KUKA KRL program: EPS_2_25694_CR02_A_20260114065854.src

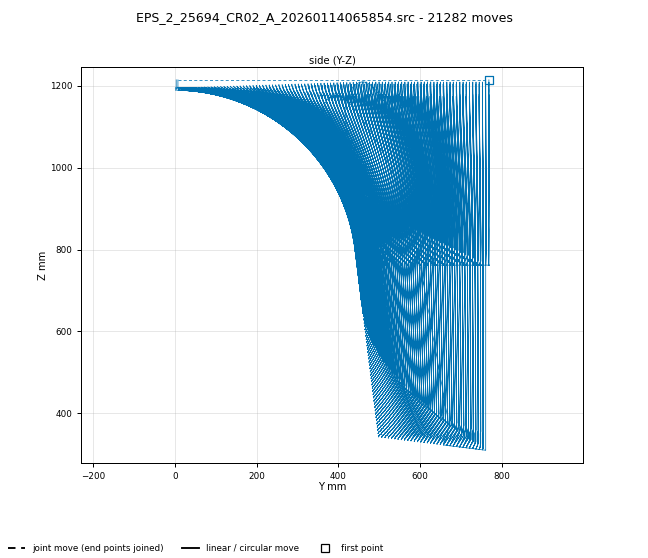
[picture p0: tool path of EPS_2_25694_CR02_A_20260114065854.src, 21282 of 21284 moves have a stored position in this frame; points joined in program order, loops and branches not executed]
&ACCESS RVP
&REL 4
&COMMENT QRS 19112012
&PARAM EDITMASK = *
DEF PART()
EXT BAS (BAS_COMMAND :IN,REAL :IN )
INT I
BAS (#INITMOV,0 )

;KUKA QRS Post kuka4.cps  Date:22-06-2017 !

File_ID=2972

QRS_PRE_INIT()

;Init var - Until changes are made in qrs_pre_init
Outlet_Square_prg=0
Inlet_1_Square_prg=0
Inlet_2_Square_prg=0
Inlet_3_Square_prg=0
Inlet_4_Square_prg=0
Inlet_5_Square_prg=0

Outlet_1={X 0.000, Y 457.000, Z 786.000, B 0.000, E1 0.000 }
Inlet_1={X 0.000, Y 457.000, Z 756.000, B 0.000, E1 180.000 }
Outlet_1_type=838
Inlet_1_type=838
;QRS#1=Sidecore dimensions
;QRS#2=825-33" Concrete
;QRS#3=825-33" Concrete
;QRS#4=
;QRS#5=
;QRS#6=
;QRS#7=
;QRS#8=
;QRS#9=S306-46
;QRS#10=S306-46
;QRS#11=
;QRS#12=
;QRS#13=
;QRS#14=
;QRS#15=
;QRS#16=1524x152x1676 5,5'
;QRS#17=EPS Height
;QRS#18=1205
;QRS#19=*
;QRS#20= UPDATED VERSION 22-06-2017
;QRS#21=*
Outlet_Square=0650
Inlet_1_Square=0650
Inlet_2_Square=0
Inlet_3_Square=0
Inlet_4_Square=0
Inlet_5_Square=0
Mill_Square=1
Outlet_Square_Prg=267
Inlet_1_Square_prg=267

QRS_INIT()

$ADVANCE=5

; T1
PTP {E1 173.011,E2 173.011}
PTP {X 0,Y 767.721,A -85,B 0,C 180,E1 173.011,E2 173.011,E3 0,E4 0,E5 0,E6 0}
QRS_SPEED_INIT()
LIN {X 0,Y 767.721,Z 1215,A -85,B 0,C 180,E1 173.011,E2 173.011,E3 0,E4 0,E5 0,E6 0} C_VEL
LIN {X 0,Y 767.721,Z 764.06,A -85,B 0,C 180,E1 173.011,E2 173.011} C_VEL
LIN {X 0,Y 767.758,Z 762.06,A -85,B 0,C 180,E1 173.16,E2 173.16} C_VEL
LIN {X 0,Y 767.849,Z 762.06,A -85,B 0,C 180,E1 173.458,E2 173.458} C_VEL
LIN {X 0,Y 767.873,Z 762.06,A -85,B 0,C 180,E1 177.201,E2 177.201} C_VEL
LIN {X 0,Y 767.866,Z 762.06,A -85,B 0,C 180,E1 180.933,E2 180.933} C_VEL
LIN {X 0,Y 767.801,Z 762.06,A -85,B 0,C 180,E1 184.668,E2 184.668} C_VEL
LIN {X 0,Y 767.796,Z 762.06,A -85,B 0,C 180,E1 188.424,E2 188.424} C_VEL
LIN {X 0,Y 767.786,Z 762.06,A -85,B 0,C 180,E1 192.216,E2 192.216} C_VEL
LIN {X 0,Y 767.853,Z 762.06,A -85,B 0,C 180,E1 196.217,E2 196.217} C_VEL
LIN {X 0,Y 767.811,Z 762.06,A -85,B 0,C 180,E1 199.987,E2 199.987} C_VEL
LIN {X 0,Y 767.795,Z 762.06,A -85,B 0,C 180,E1 204.011,E2 204.011} C_VEL
LIN {X 0,Y 767.772,Z 762.06,A -85,B 0,C 180,E1 208.166,E2 208.166} C_VEL
LIN {X 0,Y 767.321,Z 762.06,A -85,B 0,C 180,E1 210.327,E2 210.327} C_VEL
LIN {X 0,Y 767.721,Z 762.06,A -85,B 0,C 180,E1 212.492,E2 212.492} C_VEL
LIN {X 0,Y 767.405,Z 762.06,A -85,B 0,C 180,E1 213.85,E2 213.85} C_VEL
LIN {X 0,Y 767.706,Z 762.06,A -85,B 0,C 180,E1 217.097,E2 217.097} C_VEL
LIN {X 0,Y 767.171,Z 762.06,A -85,B 0,C 180,E1 220.04,E2 220.04} C_VEL
LIN {X 0,Y 767.664,Z 762.06,A -85,B 0,C 180,E1 221.871,E2 221.871} C_VEL
LIN {X 0,Y 767.687,Z 762.06,A -85,B 0,C 180,E1 222.902,E2 222.902} C_VEL
LIN {X 0,Y 767.675,Z 762.06,A -85,B 0,C 180,E1 224.427,E2 224.427} C_VEL
LIN {X 0,Y 767.633,Z 762.06,A -85,B 0,C 180,E1 225.572,E2 225.572} C_VEL
LIN {X 0,Y 767.692,Z 762.06,A -85,B 0,C 180,E1 229.916,E2 229.916} C_VEL
LIN {X 0,Y 767.75,Z 762.06,A -85,B 0,C 180,E1 230.595,E2 230.595} C_VEL
LIN {X 0,Y 767.846,Z 762.06,A -85,B 0,C 180,E1 233.563,E2 233.563} C_VEL
LIN {X 0,Y 767.229,Z 762.06,A -85,B 0,C 180,E1 233.823,E2 233.823} C_VEL
LIN {X 0,Y 766.939,Z 775.573,A -85,B 0,C 180,E1 234.02,E2 234.02} C_VEL
LIN {X 0,Y 767.282,Z 814.24,A -85,B 0,C 180,E1 234.475,E2 234.475} C_VEL
LIN {X 0,Y 767.477,Z 832.161,A -85,B 0,C 180,E1 234.718,E2 234.718} C_VEL
LIN {X 0,Y 767.376,Z 848.654,A -85,B 0,C 180,E1 234.983,E2 234.983} C_VEL
LIN {X 0,Y 767.211,Z 858.67,A -85,B 0,C 180,E1 235.166,E2 235.166} C_VEL
LIN {X 0,Y 767.33,Z 876.57,A -85,B 0,C 180,E1 235.568,E2 235.568} C_VEL
LIN {X 0,Y 767.282,Z 887.768,A -85,B 0,C 180,E1 235.85,E2 235.85} C_VEL
LIN {X 0,Y 767.451,Z 900.805,A -85,B 0,C 180,E1 236.23,E2 236.23} C_VEL
LIN {X 0,Y 767.479,Z 917.969,A -85,B 0,C 180,E1 236.766,E2 236.766} C_VEL
LIN {X 0,Y 767.395,Z 931.208,A -85,B 0,C 180,E1 237.225,E2 237.225} C_VEL
LIN {X 0,Y 767.51,Z 940.172,A -85,B 0,C 180,E1 237.569,E2 237.569} C_VEL
LIN {X 0,Y 767.582,Z 955.639,A -85,B 0,C 180,E1 238.192,E2 238.192} C_VEL
LIN {X 0,Y 767.448,Z 974.021,A -85,B 0,C 180,E1 239.005,E2 239.005} C_VEL
LIN {X 0,Y 767.587,Z 991.208,A -85,B 0,C 180,E1 239.856,E2 239.856} C_VEL
LIN {X 0,Y 767.619,Z 1008.156,A -85,B 0,C 180,E1 240.771,E2 240.771} C_VEL
LIN {X 0,Y 767.612,Z 1024.961,A -85,B 0,C 180,E1 241.762,E2 241.762} C_VEL
LIN {X 0,Y 767.627,Z 1040.382,A -85,B 0,C 180,E1 242.751,E2 242.751} C_VEL
LIN {X 0,Y 767.65,Z 1055.737,A -85,B 0,C 180,E1 243.819,E2 243.819} C_VEL
LIN {X 0,Y 767.579,Z 1070.87,A -85,B 0,C 180,E1 244.96,E2 244.96} C_VEL
LIN {X 0,Y 767.603,Z 1083.468,A -85,B 0,C 180,E1 245.983,E2 245.983} C_VEL
LIN {X 0,Y 767.694,Z 1096.523,A -85,B 0,C 180,E1 247.13,E2 247.13} C_VEL
LIN {X 0,Y 767.584,Z 1109.748,A -85,B 0,C 180,E1 248.384,E2 248.384} C_VEL
LIN {X 0,Y 767.747,Z 1122.085,A -85,B 0,C 180,E1 249.663,E2 249.663} C_VEL
LIN {X 0,Y 767.589,Z 1133.958,A -85,B 0,C 180,E1 250.998,E2 250.998} C_VEL
LIN {X 0,Y 767.631,Z 1143.982,A -85,B 0,C 180,E1 252.227,E2 252.227} C_VEL
LIN {X 0,Y 767.795,Z 1151.235,A -85,B 0,C 180,E1 253.208,E2 253.208} C_VEL
LIN {X 0,Y 767.611,Z 1156.398,A -85,B 0,C 180,E1 253.933,E2 253.933} C_VEL
LIN {X 0,Y 767.552,Z 1164.121,A -85,B 0,C 180,E1 255.094,E2 255.094} C_VEL
LIN {X 0,Y 767.84,Z 1172.641,A -85,B 0,C 180,E1 256.534,E2 256.534} C_VEL
LIN {X 0,Y 767.501,Z 1180.531,A -85,B 0,C 180,E1 258.018,E2 258.018} C_VEL
LIN {X 0,Y 767.668,Z 1187.124,A -85,B 0,C 180,E1 259.448,E2 259.448} C_VEL
LIN {X 0,Y 767.831,Z 1190.052,A -85,B 0,C 180,E1 260.16,E2 260.16} C_VEL
LIN {X 0,Y 767.523,Z 1195.334,A -85,B 0,C 180,E1 261.574,E2 261.574} C_VEL
LIN {X 0,Y 767.558,Z 1198.326,A -85,B 0,C 180,E1 262.516,E2 262.516} C_VEL
LIN {X 0,Y 767.785,Z 1200.912,A -85,B 0,C 180,E1 263.458,E2 263.458} C_VEL
LIN {X 0,Y 767.592,Z 1203.647,A -85,B 0,C 180,E1 264.582,E2 264.582} C_VEL
LIN {X 0,Y 767.51,Z 1205.161,A -85,B 0,C 180,E1 265.33,E2 265.33} C_VEL
LIN {X 0,Y 767.558,Z 1206.426,A -85,B 0,C 180,E1 266.079,E2 266.079} C_VEL
LIN {X 0,Y 767.836,Z 1207.855,A -85,B 0,C 180,E1 267.201,E2 267.201} C_VEL
LIN {X 0,Y 767.461,Z 1209.218,A -85,B 0,C 180,E1 269.067,E2 269.067} C_VEL
LIN {X 0,Y 767.845,Z 1209.143,A -85,B 0,C 180,E1 270.933,E2 270.933} C_VEL
LIN {X 0,Y 767.8,Z 1207.862,A -85,B 0,C 180,E1 272.799,E2 272.799} C_VEL
LIN {X 0,Y 767.606,Z 1206.417,A -85,B 0,C 180,E1 273.921,E2 273.921} C_VEL
LIN {X 0,Y 767.507,Z 1205.161,A -85,B 0,C 180,E1 274.67,E2 274.67} C_VEL
LIN {X 0,Y 767.614,Z 1202.789,A -85,B 0,C 180,E1 275.793,E2 275.793} C_VEL
LIN {X 0,Y 767.819,Z 1200.906,A -85,B 0,C 180,E1 276.542,E2 276.542} C_VEL
LIN {X 0,Y 767.591,Z 1198.32,A -85,B 0,C 180,E1 277.484,E2 277.484} C_VEL
LIN {X 0,Y 767.491,Z 1195.339,A -85,B 0,C 180,E1 278.427,E2 278.427} C_VEL
LIN {X 0,Y 767.749,Z 1190.065,A -85,B 0,C 180,E1 279.841,E2 279.841} C_VEL
LIN {X 0,Y 767.719,Z 1187.116,A -85,B 0,C 180,E1 280.552,E2 280.552} C_VEL
LIN {X 0,Y 767.49,Z 1179.366,A -85,B 0,C 180,E1 282.22,E2 282.22} C_VEL
LIN {X 0,Y 767.745,Z 1172.601,A -85,B 0,C 180,E1 283.477,E2 283.477} C_VEL
LIN {X 0,Y 767.714,Z 1168.739,A -85,B 0,C 180,E1 284.133,E2 284.133} C_VEL
LIN {X 0,Y 767.54,Z 1162.921,A -85,B 0,C 180,E1 285.1,E2 285.1} C_VEL
LIN {X 0,Y 767.667,Z 1153.061,A -85,B 0,C 180,E1 286.552,E2 286.552} C_VEL
LIN {X 0,Y 767.78,Z 1147.604,A -85,B 0,C 180,E1 287.28,E2 287.28} C_VEL
LIN {X 0,Y 767.63,Z 1142.008,A -85,B 0,C 180,E1 288.018,E2 288.018} C_VEL
LIN {X 0,Y 767.581,Z 1131.866,A -85,B 0,C 180,E1 289.249,E2 289.249} C_VEL
LIN {X 0,Y 767.776,Z 1119.932,A -85,B 0,C 180,E1 290.566,E2 290.566} C_VEL
LIN {X 0,Y 767.586,Z 1107.113,A -85,B 0,C 180,E1 291.872,E2 291.872} C_VEL
LIN {X 0,Y 767.666,Z 1095.113,A -85,B 0,C 180,E1 292.997,E2 292.997} C_VEL
LIN {X 0,Y 767.698,Z 1081.936,A -85,B 0,C 180,E1 294.142,E2 294.142} C_VEL
LIN {X 0,Y 767.621,Z 1067.008,A -85,B 0,C 180,E1 295.338,E2 295.338} C_VEL
LIN {X 0,Y 767.649,Z 1052.646,A -85,B 0,C 180,E1 296.401,E2 296.401} C_VEL
LIN {X 0,Y 767.608,Z 1037.373,A -85,B 0,C 180,E1 297.447,E2 297.447} C_VEL
LIN {X 0,Y 767.587,Z 1021.651,A -85,B 0,C 180,E1 298.44,E2 298.44} C_VEL
LIN {X 0,Y 767.552,Z 1006.46,A -85,B 0,C 180,E1 299.329,E2 299.329} C_VEL
LIN {X 0,Y 767.57,Z 987.929,A -85,B 0,C 180,E1 300.312,E2 300.312} C_VEL
LIN {X 0,Y 767.437,Z 969.61,A -85,B 0,C 180,E1 301.2,E2 301.2} C_VEL
LIN {X 0,Y 767.571,Z 952.399,A -85,B 0,C 180,E1 301.946,E2 301.946} C_VEL
LIN {X 0,Y 767.52,Z 932.77,A -85,B 0,C 180,E1 302.714,E2 302.714} C_VEL
LIN {X 0,Y 767.357,Z 920.452,A -85,B 0,C 180,E1 303.153,E2 303.153} C_VEL
LIN {X 0,Y 767.469,Z 911.202,A -85,B 0,C 180,E1 303.452,E2 303.452} C_VEL
LIN {X 0,Y 767.487,Z 892.927,A -85,B 0,C 180,E1 303.998,E2 303.998} C_VEL
LIN {X 0,Y 767.238,Z 876.518,A -85,B 0,C 180,E1 304.438,E2 304.438} C_VEL
LIN {X 0,Y 767.413,Z 858.66,A -85,B 0,C 180,E1 304.823,E2 304.823} C_VEL
LIN {X 0,Y 767.244,Z 840.756,A -85,B 0,C 180,E1 305.16,E2 305.16} C_VEL
LIN {X 0,Y 767.192,Z 834.749,A -85,B 0,C 180,E1 305.26,E2 305.26} C_VEL
LIN {X 0,Y 767.264,Z 817.369,A -85,B 0,C 180,E1 305.489,E2 305.489} C_VEL
LIN {X 0,Y 766.944,Z 773.119,A -85,B 0,C 180,E1 306.008,E2 306.008} C_VEL
LIN {X 0,Y 767.252,Z 762.06,A -85,B 0,C 180,E1 306.177,E2 306.177} C_VEL
LIN {X 0,Y 767.883,Z 762.06,A -85,B 0,C 180,E1 306.435,E2 306.435} C_VEL
LIN {X 0,Y 767.861,Z 762.06,A -85,B 0,C 180,E1 307.109,E2 307.109} C_VEL
LIN {X 0,Y 767.652,Z 762.06,A -85,B 0,C 180,E1 311.87,E2 311.87} C_VEL
LIN {X 0,Y 767.692,Z 762.06,A -85,B 0,C 180,E1 312.9,E2 312.9} C_VEL
LIN {X 0,Y 767.682,Z 762.06,A -85,B 0,C 180,E1 314.425,E2 314.425} C_VEL
LIN {X 0,Y 767.646,Z 762.06,A -85,B 0,C 180,E1 315.571,E2 315.571} C_VEL
LIN {X 0,Y 767.684,Z 762.06,A -85,B 0,C 180,E1 319.914,E2 319.914} C_VEL
LIN {X 0,Y 767.687,Z 762.06,A -85,B 0,C 180,E1 320.589,E2 320.589} C_VEL
LIN {X 0,Y 767.215,Z 762.06,A -85,B 0,C 180,E1 322.952,E2 322.952} C_VEL
LIN {X 0,Y 767.691,Z 762.06,A -85,B 0,C 180,E1 325.267,E2 325.267} C_VEL
LIN {X 0,Y 767.761,Z 762.06,A -85,B 0,C 180,E1 329.617,E2 329.617} C_VEL
LIN {X 0,Y 767.631,Z 762.06,A -85,B 0,C 180,E1 333.924,E2 333.924} C_VEL
LIN {X 0,Y 767.27,Z 762.06,A -85,B 0,C 180,E1 335.971,E2 335.971} C_VEL
LIN {X 0,Y 767.382,Z 762.06,A -85,B 0,C 180,E1 338.161,E2 338.161} C_VEL
LIN {X 0,Y 767.467,Z 762.06,A -85,B 0,C 180,E1 340.004,E2 340.004} C_VEL
LIN {X 0,Y 767.851,Z 762.06,A -85,B 0,C 180,E1 343.784,E2 343.784} C_VEL
LIN {X 0,Y 767.786,Z 762.06,A -85,B 0,C 180,E1 347.784,E2 347.784} C_VEL
LIN {X 0,Y 767.787,Z 762.06,A -85,B 0,C 180,E1 351.576,E2 351.576} C_VEL
LIN {X 0,Y 767.81,Z 762.06,A -85,B 0,C 180,E1 355.332,E2 355.332} C_VEL
LIN {X 0,Y 767.851,Z 762.06,A -85,B 0,C 180,E1 359.067,E2 359.067} C_VEL
LIN {X 0,Y 767.87,Z 762.06,A -85,B 0,C 180,E1 362.799,E2 362.799} C_VEL
LIN {X 0,Y 767.856,Z 762.06,A -85,B 0,C 180,E1 366.542,E2 366.542} C_VEL
LIN {X 0,Y 767.784,Z 762.06,A -85,B 0,C 180,E1 370.314,E2 370.314} C_VEL
LIN {X 0,Y 767.627,Z 762.06,A -85,B 0,C 180,E1 374.135,E2 374.135} C_VEL
LIN {X 0,Y 767.143,Z 762.06,A -85,B 0,C 180,E1 376.077,E2 376.077} C_VEL
LIN {X 0,Y 767.685,Z 762.06,A -85,B 0,C 180,E1 379.99,E2 379.99} C_VEL
LIN {X 0,Y 767.687,Z 762.06,A -85,B 0,C 180,E1 384.015,E2 384.015} C_VEL
LIN {X 0,Y 767.664,Z 762.06,A -85,B 0,C 180,E1 388.171,E2 388.171} C_VEL
LIN {X 0,Y 767.23,Z 762.06,A -85,B 0,C 180,E1 390.328,E2 390.328} C_VEL
LIN {X 0,Y 767.652,Z 762.06,A -85,B 0,C 180,E1 392.495,E2 392.495} C_VEL
LIN {X 0,Y 767.36,Z 762.06,A -85,B 0,C 180,E1 393.845,E2 393.845} C_VEL
LIN {X 0,Y 767.733,Z 762.06,A -85,B 0,C 180,E1 397.1,E2 397.1} C_VEL
LIN {X 0,Y 767.129,Z 762.06,A -85,B 0,C 180,E1 400.036,E2 400.036} C_VEL
LIN {X 0,Y 767.604,Z 762.06,A -85,B 0,C 180,E1 401.875,E2 401.875} C_VEL
LIN {X 0,Y 767.466,Z 762.06,A -85,B 0,C 180,E1 402.884,E2 402.884} C_VEL
LIN {X 0,Y 767.614,Z 762.06,A -85,B 0,C 180,E1 407.106,E2 407.106} C_VEL
LIN {X 0,Y 767.732,Z 762.06,A -85,B 0,C 180,E1 408.136,E2 408.136} C_VEL
LIN {X 0,Y 767.782,Z 762.06,A -85,B 0,C 180,E1 409.908,E2 409.908} C_VEL
LIN {X 0,Y 767.744,Z 762.06,A -85,B 0,C 180,E1 410.594,E2 410.594} C_VEL
LIN {X 0,Y 767.888,Z 762.06,A -85,B 0,C 180,E1 413.865,E2 413.865} C_VEL
LIN {X 0,Y 766.795,Z 762.06,A -85,B 0,C 180,E1 414.099,E2 414.099} C_VEL
LIN {X 0,Y 767.039,Z 764.36,A -85,B 0,C 180,E1 414.193,E2 414.193} C_VEL
LIN {X 0,Y 767.173,Z 768.976,A -85,B 0,C 180,E1 414.252,E2 414.252} C_VEL
LIN {X 0,Y 767.325,Z 796.657,A -85,B 0,C 180,E1 414.585,E2 414.585} C_VEL
LIN {X 0,Y 767.214,Z 810.558,A -85,B 0,C 180,E1 414.79,E2 414.79} C_VEL
LIN {X 0,Y 767.486,Z 827.833,A -85,B 0,C 180,E1 415.118,E2 415.118} C_VEL
LIN {X 0,Y 767.463,Z 845.793,A -85,B 0,C 180,E1 415.511,E2 415.511} C_VEL
LIN {X 0,Y 767.266,Z 858.726,A -85,B 0,C 180,E1 415.831,E2 415.831} C_VEL
LIN {X 0,Y 767.436,Z 870.934,A -85,B 0,C 180,E1 416.188,E2 416.188} C_VEL
LIN {X 0,Y 767.487,Z 888.084,A -85,B 0,C 180,E1 416.725,E2 416.725} C_VEL
LIN {X 0,Y 767.408,Z 902.504,A -85,B 0,C 180,E1 417.226,E2 417.226} C_VEL
LIN {X 0,Y 767.594,Z 923.524,A -85,B 0,C 180,E1 418.055,E2 418.055} C_VEL
LIN {X 0,Y 767.486,Z 943.55,A -85,B 0,C 180,E1 418.939,E2 418.939} C_VEL
LIN {X 0,Y 767.588,Z 960.643,A -85,B 0,C 180,E1 419.781,E2 419.781} C_VEL
LIN {X 0,Y 767.62,Z 978.565,A -85,B 0,C 180,E1 420.75,E2 420.75} C_VEL
LIN {X 0,Y 767.611,Z 994.596,A -85,B 0,C 180,E1 421.694,E2 421.694} C_VEL
LIN {X 0,Y 767.624,Z 1011.031,A -85,B 0,C 180,E1 422.751,E2 422.751} C_VEL
LIN {X 0,Y 767.646,Z 1026.339,A -85,B 0,C 180,E1 423.819,E2 423.819} C_VEL
LIN {X 0,Y 767.577,Z 1040.297,A -85,B 0,C 180,E1 424.869,E2 424.869} C_VEL
LIN {X 0,Y 767.614,Z 1053.981,A -85,B 0,C 180,E1 425.984,E2 425.984} C_VEL
LIN {X 0,Y 767.698,Z 1066.997,A -85,B 0,C 180,E1 427.13,E2 427.13} C_VEL
LIN {X 0,Y 767.592,Z 1079.52,A -85,B 0,C 180,E1 428.316,E2 428.316} C_VEL
LIN {X 0,Y 767.751,Z 1092.479,A -85,B 0,C 180,E1 429.663,E2 429.663} C_VEL
LIN {X 0,Y 767.578,Z 1103.319,A -85,B 0,C 180,E1 430.874,E2 430.874} C_VEL
LIN {X 0,Y 767.568,Z 1114.318,A -85,B 0,C 180,E1 432.226,E2 432.226} C_VEL
LIN {X 0,Y 767.794,Z 1123.389,A -85,B 0,C 180,E1 433.451,E2 433.451} C_VEL
LIN {X 0,Y 767.536,Z 1133.22,A -85,B 0,C 180,E1 434.9,E2 434.9} C_VEL
LIN {X 0,Y 767.71,Z 1141.363,A -85,B 0,C 180,E1 436.257,E2 436.257} C_VEL
LIN {X 0,Y 767.741,Z 1145.739,A -85,B 0,C 180,E1 437.067,E2 437.067} C_VEL
LIN {X 0,Y 767.557,Z 1149.599,A -85,B 0,C 180,E1 437.781,E2 437.781} C_VEL
LIN {X 0,Y 767.588,Z 1157.323,A -85,B 0,C 180,E1 439.446,E2 439.446} C_VEL
LIN {X 0,Y 767.786,Z 1160.232,A -85,B 0,C 180,E1 440.16,E2 440.16} C_VEL
LIN {X 0,Y 767.616,Z 1163.808,A -85,B 0,C 180,E1 441.103,E2 441.103} C_VEL
LIN {X 0,Y 767.506,Z 1167.008,A -85,B 0,C 180,E1 442.045,E2 442.045} C_VEL
LIN {X 0,Y 767.669,Z 1170.472,A -85,B 0,C 180,E1 443.234,E2 443.234} C_VEL
LIN {X 0,Y 767.746,Z 1172.867,A -85,B 0,C 180,E1 444.208,E2 444.208} C_VEL
LIN {X 0,Y 767.488,Z 1175.254,A -85,B 0,C 180,E1 445.33,E2 445.33} C_VEL
LIN {X 0,Y 767.468,Z 1176.517,A -85,B 0,C 180,E1 446.079,E2 446.079} C_VEL
LIN {X 0,Y 767.689,Z 1177.93,A -85,B 0,C 180,E1 447.201,E2 447.201} C_VEL
LIN {X 0,Y 767.469,Z 1179.229,A -85,B 0,C 180,E1 449.067,E2 449.067} C_VEL
LIN {X 0,Y 767.67,Z 1179.165,A -85,B 0,C 180,E1 450.933,E2 450.933} C_VEL
LIN {X 0,Y 767.56,Z 1177.86,A -85,B 0,C 180,E1 452.8,E2 452.8} C_VEL
LIN {X 0,Y 767.644,Z 1176.335,A -85,B 0,C 180,E1 453.921,E2 453.921} C_VEL
LIN {X 0,Y 767.834,Z 1175.013,A -85,B 0,C 180,E1 454.668,E2 454.668} C_VEL
LIN {X 0,Y 767.573,Z 1172.694,A -85,B 0,C 180,E1 455.793,E2 455.793} C_VEL
LIN {X 0,Y 767.549,Z 1169.56,A -85,B 0,C 180,E1 457.014,E2 457.014} C_VEL
LIN {X 0,Y 767.773,Z 1166.674,A -85,B 0,C 180,E1 457.952,E2 457.952} C_VEL
LIN {X 0,Y 767.805,Z 1165.129,A -85,B 0,C 180,E1 458.423,E2 458.423} C_VEL
LIN {X 0,Y 767.504,Z 1159.928,A -85,B 0,C 180,E1 459.844,E2 459.844} C_VEL
LIN {X 0,Y 767.556,Z 1155.871,A -85,B 0,C 180,E1 460.791,E2 460.791} C_VEL
LIN {X 0,Y 767.787,Z 1150.284,A -85,B 0,C 180,E1 461.977,E2 461.977} C_VEL
LIN {X 0,Y 767.534,Z 1141.08,A -85,B 0,C 180,E1 463.706,E2 463.706} C_VEL
LIN {X 0,Y 767.802,Z 1132.595,A -85,B 0,C 180,E1 465.095,E2 465.095} C_VEL
LIN {X 0,Y 767.54,Z 1122.732,A -85,B 0,C 180,E1 466.554,E2 466.554} C_VEL
LIN {X 0,Y 767.628,Z 1112.646,A -85,B 0,C 180,E1 467.895,E2 467.895} C_VEL
LIN {X 0,Y 767.755,Z 1104.593,A -85,B 0,C 180,E1 468.875,E2 468.875} C_VEL
LIN {X 0,Y 767.618,Z 1099.242,A -85,B 0,C 180,E1 469.496,E2 469.496} C_VEL
LIN {X 0,Y 767.576,Z 1089.784,A -85,B 0,C 180,E1 470.542,E2 470.542} C_VEL
LIN {X 0,Y 767.73,Z 1077.783,A -85,B 0,C 180,E1 471.76,E2 471.76} C_VEL
LIN {X 0,Y 767.582,Z 1064.596,A -85,B 0,C 180,E1 473,E2 473} C_VEL
LIN {X 0,Y 767.632,Z 1051.392,A -85,B 0,C 180,E1 474.143,E2 474.143} C_VEL
LIN {X 0,Y 767.668,Z 1038.114,A -85,B 0,C 180,E1 475.209,E2 475.209} C_VEL
LIN {X 0,Y 767.604,Z 1023.567,A -85,B 0,C 180,E1 476.294,E2 476.294} C_VEL
LIN {X 0,Y 767.613,Z 1007.698,A -85,B 0,C 180,E1 477.381,E2 477.381} C_VEL
LIN {X 0,Y 767.62,Z 992.088,A -85,B 0,C 180,E1 478.368,E2 478.368} C_VEL
LIN {X 0,Y 767.599,Z 975.96,A -85,B 0,C 180,E1 479.308,E2 479.308} C_VEL
LIN {X 0,Y 767.572,Z 958.73,A -85,B 0,C 180,E1 480.228,E2 480.228} C_VEL
LIN {X 0,Y 767.594,Z 940.137,A -85,B 0,C 180,E1 481.124,E2 481.124} C_VEL
LIN {X 0,Y 767.456,Z 921.256,A -85,B 0,C 180,E1 481.952,E2 481.952} C_VEL
LIN {X 0,Y 767.569,Z 905.043,A -85,B 0,C 180,E1 482.586,E2 482.586} C_VEL
LIN {X 0,Y 767.526,Z 883.788,A -85,B 0,C 180,E1 483.325,E2 483.325} C_VEL
LIN {X 0,Y 767.308,Z 869.041,A -85,B 0,C 180,E1 483.786,E2 483.786} C_VEL
LIN {X 0,Y 767.486,Z 852.178,A -85,B 0,C 180,E1 484.238,E2 484.238} C_VEL
LIN {X 0,Y 767.401,Z 835.509,A -85,B 0,C 180,E1 484.636,E2 484.636} C_VEL
LIN {X 0,Y 767.206,Z 824.123,A -85,B 0,C 180,E1 484.879,E2 484.879} C_VEL
LIN {X 0,Y 767.443,Z 807.184,A -85,B 0,C 180,E1 485.164,E2 485.164} C_VEL
LIN {X 0,Y 767.363,Z 789.381,A -85,B 0,C 180,E1 485.414,E2 485.414} C_VEL
LIN {X 0,Y 766.854,Z 762.06,A -85,B 0,C 180,E1 485.758,E2 485.758} C_VEL
LIN {X 0,Y 767.637,Z 762.06,A -85,B 0,C 180,E1 485.857,E2 485.857} C_VEL
LIN {X 0,Y 767.838,Z 762.06,A -85,B 0,C 180,E1 486.434,E2 486.434} C_VEL
LIN {X 0,Y 767.849,Z 762.06,A -85,B 0,C 180,E1 487.108,E2 487.108} C_VEL
LIN {X 0,Y 767.695,Z 762.06,A -85,B 0,C 180,E1 491.867,E2 491.867} C_VEL
LIN {X 0,Y 767.685,Z 762.06,A -85,B 0,C 180,E1 492.899,E2 492.899} C_VEL
LIN {X 0,Y 767.613,Z 762.06,A -85,B 0,C 180,E1 494.43,E2 494.43} C_VEL
LIN {X 0,Y 767.563,Z 762.06,A -85,B 0,C 180,E1 495.565,E2 495.565} C_VEL
LIN {X 0,Y 767.673,Z 762.06,A -85,B 0,C 180,E1 499.915,E2 499.915} C_VEL
LIN {X 0,Y 767.681,Z 762.06,A -85,B 0,C 180,E1 500.589,E2 500.589} C_VEL
LIN {X 0,Y 767.198,Z 762.06,A -85,B 0,C 180,E1 502.953,E2 502.953} C_VEL
LIN {X 0,Y 767.664,Z 762.06,A -85,B 0,C 180,E1 505.265,E2 505.265} C_VEL
LIN {X 0,Y 767.217,Z 762.06,A -85,B 0,C 180,E1 507.484,E2 507.484} C_VEL
LIN {X 0,Y 767.654,Z 762.06,A -85,B 0,C 180,E1 509.691,E2 509.691} C_VEL
LIN {X 0,Y 767.589,Z 762.06,A -85,B 0,C 180,E1 513.923,E2 513.923} C_VEL
LIN {X 0,Y 767.127,Z 762.06,A -85,B 0,C 180,E1 515.967,E2 515.967} C_VEL
LIN {X 0,Y 767.073,Z 762.06,A -85,B 0,C 180,E1 518.218,E2 518.218} C_VEL
LIN {X 0,Y 767.691,Z 762.06,A -85,B 0,C 180,E1 520.01,E2 520.01} C_VEL
LIN {X 0,Y 767.163,Z 762.06,A -85,B 0,C 180,E1 523.961,E2 523.961} C_VEL
LIN {X 0,Y 767.621,Z 762.06,A -85,B 0,C 180,E1 525.865,E2 525.865} C_VEL
LIN {X 0,Y 767.793,Z 762.06,A -85,B 0,C 180,E1 529.686,E2 529.686} C_VEL
LIN {X 0,Y 767.758,Z 762.06,A -85,B 0,C 180,E1 533.16,E2 533.16} C_VEL
LIN {X 0,Y 765.232,Z 762.06,A -85,B 0,C 180,E1 534.119,E2 534.119} C_VEL
LIN {X 0,Y 759.658,Z 762.06,A -85,B 0,C 180,E1 535.548,E2 535.548} C_VEL
LIN {X 0,Y 759.577,Z 762.06,A -85,B 0,C 180,E1 535.713,E2 535.713} C_VEL
LIN {X 0,Y 759.69,Z 762.06,A -85,B 0,C 180,E1 540.007,E2 540.007} C_VEL
LIN {X 0,Y 759.858,Z 762.06,A -85,B 0,C 180,E1 544.569,E2 544.569} C_VEL
LIN {X 0,Y 759.629,Z 762.06,A -85,B 0,C 180,E1 549.163,E2 549.163} C_VEL
LIN {X 0,Y 759.467,Z 762.06,A -85,B 0,C 180,E1 553.819,E2 553.819} C_VEL
LIN {X 0,Y 759.608,Z 762.06,A -85,B 0,C 180,E1 557.366,E2 557.366} C_VEL
LIN {X 0,Y 759.573,Z 762.06,A -85,B 0,C 180,E1 560.988,E2 560.988} C_VEL
LIN {X 0,Y 759.626,Z 762.06,A -85,B 0,C 180,E1 564.697,E2 564.697} C_VEL
LIN {X 0,Y 759.612,Z 762.06,A -85,B 0,C 180,E1 568.918,E2 568.918} C_VEL
LIN {X 0,Y 759.588,Z 762.06,A -85,B 0,C 180,E1 573.327,E2 573.327} C_VEL
LIN {X 0,Y 759.421,Z 762.06,A -85,B 0,C 180,E1 578.089,E2 578.089} C_VEL
LIN {X 0,Y 759.786,Z 762.06,A -85,B 0,C 180,E1 582.618,E2 582.618} C_VEL
LIN {X 0,Y 759.601,Z 762.06,A -85,B 0,C 180,E1 585.871,E2 585.871} C_VEL
LIN {X 0,Y 759.796,Z 762.06,A -85,B 0,C 180,E1 590.865,E2 590.865} C_VEL
LIN {X 0,Y 759.939,Z 762.512,A -85,B 0,C 180,E1 593.485,E2 593.485} C_VEL
LIN {X 0,Y 760.891,Z 848.299,A -85,B 0,C 180,E1 594.633,E2 594.633} C_VEL
LIN {X 0,Y 760.726,Z 894.934,A -85,B 0,C 180,E1 595.713,E2 595.713} C_VEL
LIN {X 0,Y 760.657,Z 942.42,A -85,B 0,C 180,E1 597.33,E2 597.33} C_VEL
LIN {X 0,Y 760.479,Z 988.227,A -85,B 0,C 180,E1 599.39,E2 599.39} C_VEL
LIN {X 0,Y 760.281,Z 1030.636,A -85,B 0,C 180,E1 601.832,E2 601.832} C_VEL
LIN {X 0,Y 760.109,Z 1068.915,A -85,B 0,C 180,E1 604.538,E2 604.538} C_VEL
LIN {X 0,Y 759.936,Z 1106.119,A -85,B 0,C 180,E1 607.801,E2 607.801} C_VEL
LIN {X 0,Y 759.817,Z 1135.564,A -85,B 0,C 180,E1 610.994,E2 610.994} C_VEL
LIN {X 0,Y 759.749,Z 1158.905,A -85,B 0,C 180,E1 614.128,E2 614.128} C_VEL
LIN {X 0,Y 759.745,Z 1178.001,A -85,B 0,C 180,E1 617.362,E2 617.362} C_VEL
LIN {X 0,Y 759.773,Z 1193.413,A -85,B 0,C 180,E1 620.844,E2 620.844} C_VEL
LIN {X 0,Y 759.737,Z 1203.568,A -85,B 0,C 180,E1 624.292,E2 624.292} C_VEL
LIN {X 0,Y 759.787,Z 1208.98,A -85,B 0,C 180,E1 627.72,E2 627.72} C_VEL
LIN {X 0,Y 759.929,Z 1209.669,A -85,B 0,C 180,E1 631.139,E2 631.139} C_VEL
LIN {X 0,Y 759.659,Z 1205.912,A -85,B 0,C 180,E1 634.563,E2 634.563} C_VEL
LIN {X 0,Y 759.648,Z 1197.335,A -85,B 0,C 180,E1 638.004,E2 638.004} C_VEL
LIN {X 0,Y 759.701,Z 1185.042,A -85,B 0,C 180,E1 641.182,E2 641.182} C_VEL
LIN {X 0,Y 759.752,Z 1166.459,A -85,B 0,C 180,E1 644.69,E2 644.69} C_VEL
LIN {X 0,Y 759.852,Z 1142.885,A -85,B 0,C 180,E1 648.102,E2 648.102} C_VEL
LIN {X 0,Y 759.943,Z 1112.257,A -85,B 0,C 180,E1 651.583,E2 651.583} C_VEL
LIN {X 0,Y 760.109,Z 1078.541,A -85,B 0,C 180,E1 654.675,E2 654.675} C_VEL
LIN {X 0,Y 760.274,Z 1039.4,A -85,B 0,C 180,E1 657.603,E2 657.603} C_VEL
LIN {X 0,Y 760.418,Z 995.978,A -85,B 0,C 180,E1 660.199,E2 660.199} C_VEL
LIN {X 0,Y 760.688,Z 952.908,A -85,B 0,C 180,E1 662.25,E2 662.25} C_VEL
LIN {X 0,Y 760.772,Z 906.903,A -85,B 0,C 180,E1 663.918,E2 663.918} C_VEL
LIN {X 0,Y 760.855,Z 862.847,A -85,B 0,C 180,E1 665.079,E2 665.079} C_VEL
LIN {X 0,Y 760.841,Z 817.591,A -85,B 0,C 180,E1 665.832,E2 665.832} C_VEL
LIN {X 0,Y 759.999,Z 762.06,A -85,B 0,C 180,E1 666.531,E2 666.531} C_VEL
LIN {X 0,Y 759.758,Z 762.06,A -85,B 0,C 180,E1 672.614,E2 672.614} C_VEL
LIN {X 0,Y 759.619,Z 762.06,A -85,B 0,C 180,E1 675.87,E2 675.87} C_VEL
LIN {X 0,Y 759.689,Z 762.06,A -85,B 0,C 180,E1 680.873,E2 680.873} C_VEL
LIN {X 0,Y 759.465,Z 762.06,A -85,B 0,C 180,E1 686.14,E2 686.14} C_VEL
LIN {X 0,Y 759.623,Z 762.06,A -85,B 0,C 180,E1 690.174,E2 690.174} C_VEL
LIN {X 0,Y 759.685,Z 762.06,A -85,B 0,C 180,E1 694.045,E2 694.045} C_VEL
LIN {X 0,Y 759.459,Z 762.06,A -85,B 0,C 180,E1 699.254,E2 699.254} C_VEL
LIN {X 0,Y 759.938,Z 762.06,A -85,B 0,C 180,E1 703.831,E2 703.831} C_VEL
LIN {X 0,Y 759.626,Z 762.06,A -85,B 0,C 180,E1 708.52,E2 708.52} C_VEL
LIN {X 0,Y 759.504,Z 762.06,A -85,B 0,C 180,E1 713.138,E2 713.138} C_VEL
LIN {X 0,Y 759.567,Z 762.06,A -85,B 0,C 180,E1 716.572,E2 716.572} C_VEL
LIN {X 0,Y 759.657,Z 762.06,A -85,B 0,C 180,E1 719.993,E2 719.993} C_VEL
LIN {X 0,Y 759.582,Z 762.06,A -85,B 0,C 180,E1 724.557,E2 724.557} C_VEL
LIN {X 0,Y 759.549,Z 762.06,A -85,B 0,C 180,E1 727.998,E2 727.998} C_VEL
LIN {X 0,Y 759.481,Z 762.06,A -85,B 0,C 180,E1 731.468,E2 731.468} C_VEL
LIN {X 0,Y 759.423,Z 762.06,A -85,B 0,C 180,E1 734.983,E2 734.983} C_VEL
LIN {X 0,Y 759.498,Z 762.06,A -85,B 0,C 180,E1 740.754,E2 740.754} C_VEL
LIN {X 0,Y 759.522,Z 762.06,A -85,B 0,C 180,E1 744.686,E2 744.686} C_VEL
LIN {X 0,Y 759.522,Z 762.06,A -85,B 0,C 180,E1 748.908,E2 748.908} C_VEL
LIN {X 0,Y 759.526,Z 762.06,A -85,B 0,C 180,E1 753.322,E2 753.322} C_VEL
LIN {X 0,Y 759.428,Z 762.06,A -85,B 0,C 180,E1 758.072,E2 758.072} C_VEL
LIN {X 0,Y 759.587,Z 762.06,A -85,B 0,C 180,E1 762.603,E2 762.603} C_VEL
LIN {X 0,Y 759.727,Z 762.06,A -85,B 0,C 180,E1 767.448,E2 767.448} C_VEL
LIN {X 0,Y 759.615,Z 762.06,A -85,B 0,C 180,E1 771.926,E2 771.926} C_VEL
LIN {X 0,Y 759.953,Z 762.06,A -85,B 0,C 180,E1 773.771,E2 773.771} C_VEL
LIN {X 0,Y 760.8,Z 807.354,A -85,B 0,C 180,E1 774.395,E2 774.395} C_VEL
LIN {X 0,Y 760.69,Z 858.035,A -85,B 0,C 180,E1 775.475,E2 775.475} C_VEL
LIN {X 0,Y 760.617,Z 906.695,A -85,B 0,C 180,E1 777.054,E2 777.054} C_VEL
LIN {X 0,Y 760.473,Z 954.122,A -85,B 0,C 180,E1 779.143,E2 779.143} C_VEL
LIN {X 0,Y 760.308,Z 996.347,A -85,B 0,C 180,E1 781.511,E2 781.511} C_VEL
LIN {X 0,Y 760.104,Z 1038.487,A -85,B 0,C 180,E1 784.46,E2 784.46} C_VEL
LIN {X 0,Y 759.952,Z 1074.991,A -85,B 0,C 180,E1 787.649,E2 787.649} C_VEL
LIN {X 0,Y 759.832,Z 1104.719,A -85,B 0,C 180,E1 790.845,E2 790.845} C_VEL
LIN {X 0,Y 759.781,Z 1129.213,A -85,B 0,C 180,E1 794.13,E2 794.13} C_VEL
LIN {X 0,Y 759.812,Z 1148.246,A -85,B 0,C 180,E1 797.364,E2 797.364} C_VEL
LIN {X 0,Y 759.798,Z 1163.575,A -85,B 0,C 180,E1 800.846,E2 800.846} C_VEL
LIN {X 0,Y 759.855,Z 1173.672,A -85,B 0,C 180,E1 804.294,E2 804.294} C_VEL
LIN {X 0,Y 759.688,Z 1179.017,A -85,B 0,C 180,E1 807.721,E2 807.721} C_VEL
LIN {X 0,Y 759.747,Z 1179.655,A -85,B 0,C 180,E1 811.14,E2 811.14} C_VEL
LIN {X 0,Y 759.948,Z 1175.828,A -85,B 0,C 180,E1 814.563,E2 814.563} C_VEL
LIN {X 0,Y 759.931,Z 1167.188,A -85,B 0,C 180,E1 818.002,E2 818.002} C_VEL
LIN {X 0,Y 759.853,Z 1152.127,A -85,B 0,C 180,E1 821.762,E2 821.762} C_VEL
LIN {X 0,Y 759.939,Z 1132.553,A -85,B 0,C 180,E1 825.277,E2 825.277} C_VEL
LIN {X 0,Y 759.979,Z 1105.2,A -85,B 0,C 180,E1 829.002,E2 829.002} C_VEL
LIN {X 0,Y 760.005,Z 1075.647,A -85,B 0,C 180,E1 832.197,E2 832.197} C_VEL
LIN {X 0,Y 760.163,Z 1040.303,A -85,B 0,C 180,E1 835.303,E2 835.303} C_VEL
LIN {X 0,Y 760.291,Z 999.939,A -85,B 0,C 180,E1 838.168,E2 838.168} C_VEL
LIN {X 0,Y 760.505,Z 958.993,A -85,B 0,C 180,E1 840.526,E2 840.526} C_VEL
LIN {X 0,Y 760.642,Z 912.875,A -85,B 0,C 180,E1 842.608,E2 842.608} C_VEL
LIN {X 0,Y 760.757,Z 865.642,A -85,B 0,C 180,E1 844.221,E2 844.221} C_VEL
LIN {X 0,Y 760.847,Z 817.475,A -85,B 0,C 180,E1 845.34,E2 845.34} C_VEL
LIN {X 0,Y 759.844,Z 762.486,A -85,B 0,C 180,E1 846.131,E2 846.131} C_VEL
LIN {X 0,Y 759.468,Z 762.06,A -85,B 0,C 180,E1 851.042,E2 851.042} C_VEL
LIN {X 0,Y 759.717,Z 762.06,A -85,B 0,C 180,E1 854.287,E2 854.287} C_VEL
LIN {X 0,Y 759.667,Z 762.06,A -85,B 0,C 180,E1 860.877,E2 860.877} C_VEL
LIN {X 0,Y 759.459,Z 762.06,A -85,B 0,C 180,E1 866.156,E2 866.156} C_VEL
LIN {X 0,Y 759.548,Z 762.06,A -85,B 0,C 180,E1 870.186,E2 870.186} C_VEL
LIN {X 0,Y 759.65,Z 762.06,A -85,B 0,C 180,E1 874.058,E2 874.058} C_VEL
LIN {X 0,Y 759.652,Z 762.06,A -85,B 0,C 180,E1 880.244,E2 880.244} C_VEL
LIN {X 0,Y 759.617,Z 762.06,A -85,B 0,C 180,E1 886.198,E2 886.198} C_VEL
LIN {X 0,Y 759.567,Z 762.06,A -85,B 0,C 180,E1 890.85,E2 890.85} C_VEL
LIN {X 0,Y 759.691,Z 762.06,A -85,B 0,C 180,E1 894.3,E2 894.3} C_VEL
LIN {X 0,Y 759.577,Z 762.06,A -85,B 0,C 180,E1 895.713,E2 895.713} C_VEL
LIN {X 0,Y 755.755,Z 762.06,A -85,B 0,C 180,E1 897.001,E2 897.001} C_VEL
LIN {X 0,Y 751.74,Z 762.06,A -85,B 0,C 180,E1 898.303,E2 898.303} C_VEL
LIN {X 0,Y 751.688,Z 762.06,A -85,B 0,C 180,E1 902.311,E2 902.311} C_VEL
LIN {X 0,Y 751.684,Z 762.06,A -85,B 0,C 180,E1 905.775,E2 905.775} C_VEL
LIN {X 0,Y 751.603,Z 762.06,A -85,B 0,C 180,E1 909.882,E2 909.882} C_VEL
LIN {X 0,Y 751.563,Z 762.06,A -85,B 0,C 180,E1 913.967,E2 913.967} C_VEL
LIN {X 0,Y 751.678,Z 762.06,A -85,B 0,C 180,E1 917.555,E2 917.555} C_VEL
LIN {X 0,Y 751.626,Z 762.06,A -85,B 0,C 180,E1 921.22,E2 921.22} C_VEL
LIN {X 0,Y 751.606,Z 762.06,A -85,B 0,C 180,E1 925.212,E2 925.212} C_VEL
LIN {X 0,Y 751.55,Z 762.06,A -85,B 0,C 180,E1 930.164,E2 930.164} C_VEL
LIN {X 0,Y 751.812,Z 762.06,A -85,B 0,C 180,E1 932.87,E2 932.87} C_VEL
LIN {X 0,Y 751.784,Z 762.06,A -85,B 0,C 180,E1 937.089,E2 937.089} C_VEL
LIN {X 0,Y 751.826,Z 762.06,A -85,B 0,C 180,E1 943.11,E2 943.11} C_VEL
LIN {X 0,Y 751.412,Z 762.06,A -85,B 0,C 180,E1 946.862,E2 946.862} C_VEL
LIN {X 0,Y 751.769,Z 762.06,A -85,B 0,C 180,E1 951.623,E2 951.623} C_VEL
LIN {X 0,Y 751.912,Z 762.371,A -85,B 0,C 180,E1 953.029,E2 953.029} C_VEL
LIN {X 0,Y 754.166,Z 769.226,A -85,B 0,C 180,E1 953.238,E2 953.238} C_VEL
LIN {X 0,Y 754.438,Z 847.508,A -85,B 0,C 180,E1 954.269,E2 954.269} C_VEL
LIN {X 0,Y 754.064,Z 893.687,A -85,B 0,C 180,E1 955.332,E2 955.332} C_VEL
LIN {X 0,Y 753.786,Z 940.821,A -85,B 0,C 180,E1 956.929,E2 956.929} C_VEL
LIN {X 0,Y 753.404,Z 987.353,A -85,B 0,C 180,E1 959.027,E2 959.027} C_VEL
LIN {X 0,Y 753.006,Z 1029.302,A -85,B 0,C 180,E1 961.448,E2 961.448} C_VEL
LIN {X 0,Y 752.646,Z 1069.034,A -85,B 0,C 180,E1 964.276,E2 964.276} C_VEL
LIN {X 0,Y 752.317,Z 1106.12,A -85,B 0,C 180,E1 967.564,E2 967.564} C_VEL
LIN {X 0,Y 752.073,Z 1135.607,A -85,B 0,C 180,E1 970.795,E2 970.795} C_VEL
LIN {X 0,Y 751.931,Z 1160.77,A -85,B 0,C 180,E1 974.241,E2 974.241} C_VEL
LIN {X 0,Y 751.859,Z 1179.553,A -85,B 0,C 180,E1 977.522,E2 977.522} C_VEL
LIN {X 0,Y 751.835,Z 1194.428,A -85,B 0,C 180,E1 981.038,E2 981.038} C_VEL
LIN {X 0,Y 751.86,Z 1203.568,A -85,B 0,C 180,E1 984.232,E2 984.232} C_VEL
LIN {X 0,Y 751.887,Z 1208.977,A -85,B 0,C 180,E1 987.696,E2 987.696} C_VEL
LIN {X 0,Y 752.027,Z 1209.669,A -85,B 0,C 180,E1 991.151,E2 991.151} C_VEL
LIN {X 0,Y 751.768,Z 1205.912,A -85,B 0,C 180,E1 994.611,E2 994.611} C_VEL
LIN {X 0,Y 751.748,Z 1197.335,A -85,B 0,C 180,E1 998.088,E2 998.088} C_VEL
LIN {X 0,Y 751.819,Z 1185.044,A -85,B 0,C 180,E1 1001.301,E2 1001.301} C_VEL
LIN {X 0,Y 751.899,Z 1166.46,A -85,B 0,C 180,E1 1004.846,E2 1004.846} C_VEL
LIN {X 0,Y 752.036,Z 1142.884,A -85,B 0,C 180,E1 1008.298,E2 1008.298} C_VEL
LIN {X 0,Y 752.245,Z 1112.259,A -85,B 0,C 180,E1 1011.815,E2 1011.815} C_VEL
LIN {X 0,Y 752.572,Z 1078.541,A -85,B 0,C 180,E1 1014.939,E2 1014.939} C_VEL
LIN {X 0,Y 752.944,Z 1039.147,A -85,B 0,C 180,E1 1017.912,E2 1017.912} C_VEL
LIN {X 0,Y 753.336,Z 994.926,A -85,B 0,C 180,E1 1020.571,E2 1020.571} C_VEL
LIN {X 0,Y 753.823,Z 951.968,A -85,B 0,C 180,E1 1022.618,E2 1022.618} C_VEL
LIN {X 0,Y 754.099,Z 906.549,A -85,B 0,C 180,E1 1024.271,E2 1024.271} C_VEL
LIN {X 0,Y 754.343,Z 863.678,A -85,B 0,C 180,E1 1025.41,E2 1025.41} C_VEL
LIN {X 0,Y 754.415,Z 817.83,A -85,B 0,C 180,E1 1026.182,E2 1026.182} C_VEL
LIN {X 0,Y 753.606,Z 766.774,A -85,B 0,C 180,E1 1026.822,E2 1026.822} C_VEL
LIN {X 0,Y 752.022,Z 762.06,A -85,B 0,C 180,E1 1026.998,E2 1026.998} C_VEL
LIN {X 0,Y 751.81,Z 762.06,A -85,B 0,C 180,E1 1033.108,E2 1033.108} C_VEL
LIN {X 0,Y 751.409,Z 762.06,A -85,B 0,C 180,E1 1036.86,E2 1036.86} C_VEL
LIN {X 0,Y 751.606,Z 762.06,A -85,B 0,C 180,E1 1041.443,E2 1041.443} C_VEL
LIN {X 0,Y 751.556,Z 762.06,A -85,B 0,C 180,E1 1045.735,E2 1045.735} C_VEL
LIN {X 0,Y 751.68,Z 762.06,A -85,B 0,C 180,E1 1049.826,E2 1049.826} C_VEL
LIN {X 0,Y 751.52,Z 762.06,A -85,B 0,C 180,E1 1055.019,E2 1055.019} C_VEL
LIN {X 0,Y 751.577,Z 762.06,A -85,B 0,C 180,E1 1060.009,E2 1060.009} C_VEL
LIN {X 0,Y 751.699,Z 762.06,A -85,B 0,C 180,E1 1064.846,E2 1064.846} C_VEL
LIN {X 0,Y 751.614,Z 762.06,A -85,B 0,C 180,E1 1069.57,E2 1069.57} C_VEL
LIN {X 0,Y 751.685,Z 762.06,A -85,B 0,C 180,E1 1074.225,E2 1074.225} C_VEL
LIN {X 0,Y 751.955,Z 762.06,A -85,B 0,C 180,E1 1078.842,E2 1078.842} C_VEL
LIN {X 0,Y 751.868,Z 762.06,A -85,B 0,C 180,E1 1083.45,E2 1083.45} C_VEL
LIN {X 0,Y 751.64,Z 762.06,A -85,B 0,C 180,E1 1088.082,E2 1088.082} C_VEL
LIN {X 0,Y 751.556,Z 762.06,A -85,B 0,C 180,E1 1091.591,E2 1091.591} C_VEL
LIN {X 0,Y 751.472,Z 762.06,A -85,B 0,C 180,E1 1095.159,E2 1095.159} C_VEL
LIN {X 0,Y 751.698,Z 762.06,A -85,B 0,C 180,E1 1099.973,E2 1099.973} C_VEL
LIN {X 0,Y 751.535,Z 762.06,A -85,B 0,C 180,E1 1104.966,E2 1104.966} C_VEL
LIN {X 0,Y 751.637,Z 762.06,A -85,B 0,C 180,E1 1108.837,E2 1108.837} C_VEL
LIN {X 0,Y 751.755,Z 762.06,A -85,B 0,C 180,E1 1112.857,E2 1112.857} C_VEL
LIN {X 0,Y 751.803,Z 762.06,A -85,B 0,C 180,E1 1117.071,E2 1117.071} C_VEL
LIN {X 0,Y 751.508,Z 762.06,A -85,B 0,C 180,E1 1123.115,E2 1123.115} C_VEL
LIN {X 0,Y 751.801,Z 762.06,A -85,B 0,C 180,E1 1128.449,E2 1128.449} C_VEL
LIN {X 0,Y 751.913,Z 762.06,A -85,B 0,C 180,E1 1133.325,E2 1133.325} C_VEL
LIN {X 0,Y 754.331,Z 769.301,A -85,B 0,C 180,E1 1133.552,E2 1133.552} C_VEL
LIN {X 0,Y 754.41,Z 822.943,A -85,B 0,C 180,E1 1134.327,E2 1134.327} C_VEL
LIN {X 0,Y 754.071,Z 869.671,A -85,B 0,C 180,E1 1135.466,E2 1135.466} C_VEL
LIN {X 0,Y 753.76,Z 918.101,A -85,B 0,C 180,E1 1137.178,E2 1137.178} C_VEL
LIN {X 0,Y 753.397,Z 960.906,A -85,B 0,C 180,E1 1139.166,E2 1139.166} C_VEL
LIN {X 0,Y 752.973,Z 1005.217,A -85,B 0,C 180,E1 1141.788,E2 1141.788} C_VEL
LIN {X 0,Y 752.532,Z 1043.617,A -85,B 0,C 180,E1 1144.607,E2 1144.607} C_VEL
LIN {X 0,Y 752.301,Z 1078.207,A -85,B 0,C 180,E1 1147.721,E2 1147.721} C_VEL
LIN {X 0,Y 752.017,Z 1107.613,A -85,B 0,C 180,E1 1151,E2 1151} C_VEL
LIN {X 0,Y 751.948,Z 1131.268,A -85,B 0,C 180,E1 1154.272,E2 1154.272} C_VEL
LIN {X 0,Y 751.92,Z 1149.795,A -85,B 0,C 180,E1 1157.524,E2 1157.524} C_VEL
LIN {X 0,Y 751.862,Z 1164.588,A -85,B 0,C 180,E1 1161.04,E2 1161.04} C_VEL
LIN {X 0,Y 751.953,Z 1173.671,A -85,B 0,C 180,E1 1164.234,E2 1164.234} C_VEL
LIN {X 0,Y 751.785,Z 1179.017,A -85,B 0,C 180,E1 1167.697,E2 1167.697} C_VEL
LIN {X 0,Y 751.844,Z 1179.655,A -85,B 0,C 180,E1 1171.152,E2 1171.152} C_VEL
LIN {X 0,Y 752.036,Z 1175.829,A -85,B 0,C 180,E1 1174.611,E2 1174.611} C_VEL
LIN {X 0,Y 752.026,Z 1167.189,A -85,B 0,C 180,E1 1178.086,E2 1178.086} C_VEL
LIN {X 0,Y 752.01,Z 1152.13,A -85,B 0,C 180,E1 1181.887,E2 1181.887} C_VEL
LIN {X 0,Y 752.026,Z 1131.835,A -85,B 0,C 180,E1 1185.551,E2 1185.551} C_VEL
LIN {X 0,Y 752.206,Z 1104.664,A -85,B 0,C 180,E1 1189.274,E2 1189.274} C_VEL
LIN {X 0,Y 752.345,Z 1074.69,A -85,B 0,C 180,E1 1192.528,E2 1192.528} C_VEL
LIN {X 0,Y 752.701,Z 1038.127,A -85,B 0,C 180,E1 1195.747,E2 1195.747} C_VEL
LIN {X 0,Y 753.054,Z 996.731,A -85,B 0,C 180,E1 1198.673,E2 1198.673} C_VEL
LIN {X 0,Y 753.456,Z 954.729,A -85,B 0,C 180,E1 1201.056,E2 1201.056} C_VEL
LIN {X 0,Y 753.843,Z 909.416,A -85,B 0,C 180,E1 1203.08,E2 1203.08} C_VEL
LIN {X 0,Y 754.189,Z 862.766,A -85,B 0,C 180,E1 1204.642,E2 1204.642} C_VEL
LIN {X 0,Y 754.433,Z 815.808,A -85,B 0,C 180,E1 1205.717,E2 1205.717} C_VEL
LIN {X 0,Y 753.492,Z 766.628,A -85,B 0,C 180,E1 1206.436,E2 1206.436} C_VEL
LIN {X 0,Y 752.063,Z 762.06,A -85,B 0,C 180,E1 1206.633,E2 1206.633} C_VEL
LIN {X 0,Y 751.812,Z 762.06,A -85,B 0,C 180,E1 1213.11,E2 1213.11} C_VEL
LIN {X 0,Y 751.343,Z 762.06,A -85,B 0,C 180,E1 1216.874,E2 1216.874} C_VEL
LIN {X 0,Y 751.583,Z 762.06,A -85,B 0,C 180,E1 1221.458,E2 1221.458} C_VEL
LIN {X 0,Y 751.544,Z 762.06,A -85,B 0,C 180,E1 1225.75,E2 1225.75} C_VEL
LIN {X 0,Y 751.605,Z 762.06,A -85,B 0,C 180,E1 1229.838,E2 1229.838} C_VEL
LIN {X 0,Y 751.424,Z 762.06,A -85,B 0,C 180,E1 1235.03,E2 1235.03} C_VEL
LIN {X 0,Y 751.689,Z 762.06,A -85,B 0,C 180,E1 1240.026,E2 1240.026} C_VEL
LIN {X 0,Y 751.676,Z 762.06,A -85,B 0,C 180,E1 1246.049,E2 1246.049} C_VEL
LIN {X 0,Y 751.685,Z 762.06,A -85,B 0,C 180,E1 1250.753,E2 1250.753} C_VEL
LIN {X 0,Y 751.818,Z 762.06,A -85,B 0,C 180,E1 1254.24,E2 1254.24} C_VEL
LIN {X 0,Y 751.74,Z 762.06,A -85,B 0,C 180,E1 1258.303,E2 1258.303} C_VEL
LIN {X 0,Y 747.747,Z 762.06,A -85,B 0,C 180,E1 1259.609,E2 1259.609} C_VEL
LIN {X 0,Y 744.016,Z 762.06,A -85,B 0,C 180,E1 1260.929,E2 1260.929} C_VEL
LIN {X 0,Y 743.793,Z 762.06,A -85,B 0,C 180,E1 1265.836,E2 1265.836} C_VEL
LIN {X 0,Y 743.71,Z 762.06,A -85,B 0,C 180,E1 1270.542,E2 1270.542} C_VEL
LIN {X 0,Y 743.843,Z 762.06,A -85,B 0,C 180,E1 1275.318,E2 1275.318} C_VEL
LIN {X 0,Y 743.925,Z 762.06,A -85,B 0,C 180,E1 1280.206,E2 1280.206} C_VEL
LIN {X 0,Y 743.726,Z 762.06,A -85,B 0,C 180,E1 1285.261,E2 1285.261} C_VEL
LIN {X 0,Y 743.763,Z 762.06,A -85,B 0,C 180,E1 1289.187,E2 1289.187} C_VEL
LIN {X 0,Y 743.735,Z 762.06,A -85,B 0,C 180,E1 1293.587,E2 1293.587} C_VEL
LIN {X 0,Y 743.716,Z 762.06,A -85,B 0,C 180,E1 1297.587,E2 1297.587} C_VEL
LIN {X 0,Y 743.906,Z 762.06,A -85,B 0,C 180,E1 1303.006,E2 1303.006} C_VEL
LIN {X 0,Y 743.512,Z 762.06,A -85,B 0,C 180,E1 1307.028,E2 1307.028} C_VEL
LIN {X 0,Y 743.82,Z 762.06,A -85,B 0,C 180,E1 1310.965,E2 1310.965} C_VEL
LIN {X 0,Y 743.934,Z 762.781,A -85,B 0,C 180,E1 1312.57,E2 1312.57} C_VEL
LIN {X 0,Y 747.827,Z 771.806,A -85,B 0,C 180,E1 1312.905,E2 1312.905} C_VEL
LIN {X 0,Y 748.025,Z 847.074,A -85,B 0,C 180,E1 1313.908,E2 1313.908} C_VEL
LIN {X 0,Y 747.433,Z 892.946,A -85,B 0,C 180,E1 1314.959,E2 1314.959} C_VEL
LIN {X 0,Y 747,Z 940.209,A -85,B 0,C 180,E1 1316.564,E2 1316.564} C_VEL
LIN {X 0,Y 746.372,Z 986.798,A -85,B 0,C 180,E1 1318.675,E2 1318.675} C_VEL
LIN {X 0,Y 745.783,Z 1028.705,A -85,B 0,C 180,E1 1321.106,E2 1321.106} C_VEL
LIN {X 0,Y 745.191,Z 1069.544,A -85,B 0,C 180,E1 1324.042,E2 1324.042} C_VEL
LIN {X 0,Y 744.686,Z 1106.122,A -85,B 0,C 180,E1 1327.322,E2 1327.322} C_VEL
LIN {X 0,Y 744.346,Z 1135.609,A -85,B 0,C 180,E1 1330.588,E2 1330.588} C_VEL
LIN {X 0,Y 744.103,Z 1160.883,A -85,B 0,C 180,E1 1334.088,E2 1334.088} C_VEL
LIN {X 0,Y 744.02,Z 1179.61,A -85,B 0,C 180,E1 1337.399,E2 1337.399} C_VEL
LIN {X 0,Y 743.991,Z 1194.428,A -85,B 0,C 180,E1 1340.943,E2 1340.943} C_VEL
LIN {X 0,Y 743.933,Z 1204.176,A -85,B 0,C 180,E1 1344.444,E2 1344.444} C_VEL
LIN {X 0,Y 743.985,Z 1208.974,A -85,B 0,C 180,E1 1347.671,E2 1347.671} C_VEL
LIN {X 0,Y 744.125,Z 1209.669,A -85,B 0,C 180,E1 1351.163,E2 1351.163} C_VEL
LIN {X 0,Y 743.867,Z 1205.912,A -85,B 0,C 180,E1 1354.66,E2 1354.66} C_VEL
LIN {X 0,Y 743.849,Z 1197.335,A -85,B 0,C 180,E1 1358.175,E2 1358.175} C_VEL
LIN {X 0,Y 743.929,Z 1185.045,A -85,B 0,C 180,E1 1361.422,E2 1361.422} C_VEL
LIN {X 0,Y 744.067,Z 1166.462,A -85,B 0,C 180,E1 1365.006,E2 1365.006} C_VEL
LIN {X 0,Y 744.249,Z 1144.068,A -85,B 0,C 180,E1 1368.343,E2 1368.343} C_VEL
LIN {X 0,Y 744.585,Z 1115.351,A -85,B 0,C 180,E1 1371.723,E2 1371.723} C_VEL
LIN {X 0,Y 745.039,Z 1082.247,A -85,B 0,C 180,E1 1374.899,E2 1374.899} C_VEL
LIN {X 0,Y 745.614,Z 1041.479,A -85,B 0,C 180,E1 1378.045,E2 1378.045} C_VEL
LIN {X 0,Y 746.172,Z 1001.419,A -85,B 0,C 180,E1 1380.535,E2 1380.535} C_VEL
LIN {X 0,Y 746.814,Z 957.597,A -85,B 0,C 180,E1 1382.713,E2 1382.713} C_VEL
LIN {X 0,Y 747.39,Z 914.031,A -85,B 0,C 180,E1 1384.385,E2 1384.385} C_VEL
LIN {X 0,Y 747.802,Z 867.484,A -85,B 0,C 180,E1 1385.681,E2 1385.681} C_VEL
LIN {X 0,Y 748.026,Z 821.177,A -85,B 0,C 180,E1 1386.498,E2 1386.498} C_VEL
LIN {X 0,Y 747.363,Z 770.064,A -85,B 0,C 180,E1 1387.143,E2 1387.143} C_VEL
LIN {X 0,Y 743.909,Z 762.06,A -85,B 0,C 180,E1 1387.467,E2 1387.467} C_VEL
LIN {X 0,Y 743.908,Z 762.06,A -85,B 0,C 180,E1 1393.681,E2 1393.681} C_VEL
LIN {X 0,Y 743.525,Z 762.06,A -85,B 0,C 180,E1 1398.761,E2 1398.761} C_VEL
LIN {X 0,Y 743.534,Z 762.06,A -85,B 0,C 180,E1 1402.429,E2 1402.429} C_VEL
LIN {X 0,Y 743.512,Z 762.06,A -85,B 0,C 180,E1 1406.716,E2 1406.716} C_VEL
LIN {X 0,Y 743.56,Z 762.06,A -85,B 0,C 180,E1 1410.911,E2 1410.911} C_VEL
LIN {X 0,Y 743.689,Z 762.06,A -85,B 0,C 180,E1 1414.738,E2 1414.738} C_VEL
LIN {X 0,Y 743.639,Z 762.06,A -85,B 0,C 180,E1 1419.786,E2 1419.786} C_VEL
LIN {X 0,Y 743.848,Z 762.06,A -85,B 0,C 180,E1 1424.682,E2 1424.682} C_VEL
LIN {X 0,Y 743.712,Z 762.06,A -85,B 0,C 180,E1 1429.458,E2 1429.458} C_VEL
LIN {X 0,Y 743.788,Z 762.06,A -85,B 0,C 180,E1 1434.164,E2 1434.164} C_VEL
LIN {X 0,Y 744.048,Z 762.06,A -85,B 0,C 180,E1 1438.83,E2 1438.83} C_VEL
LIN {X 0,Y 743.957,Z 762.06,A -85,B 0,C 180,E1 1443.486,E2 1443.486} C_VEL
LIN {X 0,Y 743.733,Z 762.06,A -85,B 0,C 180,E1 1448.169,E2 1448.169} C_VEL
LIN {X 0,Y 743.637,Z 762.06,A -85,B 0,C 180,E1 1451.716,E2 1451.716} C_VEL
LIN {X 0,Y 743.555,Z 762.06,A -85,B 0,C 180,E1 1455.31,E2 1455.31} C_VEL
LIN {X 0,Y 743.636,Z 762.06,A -85,B 0,C 180,E1 1460.814,E2 1460.814} C_VEL
LIN {X 0,Y 743.59,Z 762.06,A -85,B 0,C 180,E1 1465.251,E2 1465.251} C_VEL
LIN {X 0,Y 743.664,Z 762.06,A -85,B 0,C 180,E1 1469.176,E2 1469.176} C_VEL
LIN {X 0,Y 743.682,Z 762.06,A -85,B 0,C 180,E1 1473.583,E2 1473.583} C_VEL
LIN {X 0,Y 743.713,Z 762.06,A -85,B 0,C 180,E1 1477.589,E2 1477.589} C_VEL
LIN {X 0,Y 743.615,Z 762.06,A -85,B 0,C 180,E1 1482.983,E2 1482.983} C_VEL
LIN {X 0,Y 743.898,Z 762.06,A -85,B 0,C 180,E1 1488.71,E2 1488.71} C_VEL
LIN {X 0,Y 743.903,Z 762.06,A -85,B 0,C 180,E1 1492.846,E2 1492.846} C_VEL
LIN {X 0,Y 748.004,Z 771.519,A -85,B 0,C 180,E1 1493.22,E2 1493.22} C_VEL
LIN {X 0,Y 747.952,Z 823.253,A -85,B 0,C 180,E1 1493.977,E2 1493.977} C_VEL
LIN {X 0,Y 747.423,Z 871.259,A -85,B 0,C 180,E1 1495.166,E2 1495.166} C_VEL
LIN {X 0,Y 746.907,Z 919.367,A -85,B 0,C 180,E1 1496.89,E2 1496.89} C_VEL
LIN {X 0,Y 746.339,Z 962.239,A -85,B 0,C 180,E1 1498.916,E2 1498.916} C_VEL
LIN {X 0,Y 745.663,Z 1006.717,A -85,B 0,C 180,E1 1501.585,E2 1501.585} C_VEL
LIN {X 0,Y 745.027,Z 1045.091,A -85,B 0,C 180,E1 1504.457,E2 1504.457} C_VEL
LIN {X 0,Y 744.631,Z 1079.884,A -85,B 0,C 180,E1 1507.652,E2 1507.652} C_VEL
LIN {X 0,Y 744.237,Z 1109.588,A -85,B 0,C 180,E1 1511.043,E2 1511.043} C_VEL
LIN {X 0,Y 744.105,Z 1133.872,A -85,B 0,C 180,E1 1514.506,E2 1514.506} C_VEL
LIN {X 0,Y 743.938,Z 1152.548,A -85,B 0,C 180,E1 1517.984,E2 1517.984} C_VEL
LIN {X 0,Y 743.966,Z 1165.602,A -85,B 0,C 180,E1 1521.238,E2 1521.238} C_VEL
LIN {X 0,Y 743.942,Z 1174.919,A -85,B 0,C 180,E1 1524.774,E2 1524.774} C_VEL
LIN {X 0,Y 743.882,Z 1179.015,A -85,B 0,C 180,E1 1527.672,E2 1527.672} C_VEL
LIN {X 0,Y 743.941,Z 1179.655,A -85,B 0,C 180,E1 1531.164,E2 1531.164} C_VEL
LIN {X 0,Y 744.126,Z 1175.83,A -85,B 0,C 180,E1 1534.66,E2 1534.66} C_VEL
LIN {X 0,Y 744.118,Z 1167.19,A -85,B 0,C 180,E1 1538.173,E2 1538.173} C_VEL
LIN {X 0,Y 744.131,Z 1152.134,A -85,B 0,C 180,E1 1542.014,E2 1542.014} C_VEL
LIN {X 0,Y 744.176,Z 1131.766,A -85,B 0,C 180,E1 1545.73,E2 1545.73} C_VEL
LIN {X 0,Y 744.433,Z 1104.67,A -85,B 0,C 180,E1 1549.483,E2 1549.483} C_VEL
LIN {X 0,Y 744.709,Z 1074.697,A -85,B 0,C 180,E1 1552.772,E2 1552.772} C_VEL
LIN {X 0,Y 745.251,Z 1038.602,A -85,B 0,C 180,E1 1555.987,E2 1555.987} C_VEL
LIN {X 0,Y 745.836,Z 996.444,A -85,B 0,C 180,E1 1558.997,E2 1558.997} C_VEL
LIN {X 0,Y 746.459,Z 953.979,A -85,B 0,C 180,E1 1561.419,E2 1561.419} C_VEL
LIN {X 0,Y 747.086,Z 908.671,A -85,B 0,C 180,E1 1563.449,E2 1563.449} C_VEL
LIN {X 0,Y 747.609,Z 862.789,A -85,B 0,C 180,E1 1564.991,E2 1564.991} C_VEL
LIN {X 0,Y 747.971,Z 816.979,A -85,B 0,C 180,E1 1566.052,E2 1566.052} C_VEL
LIN {X 0,Y 747.181,Z 769.772,A -85,B 0,C 180,E1 1566.758,E2 1566.758} C_VEL
LIN {X 0,Y 744.058,Z 762.06,A -85,B 0,C 180,E1 1567.069,E2 1567.069} C_VEL
LIN {X 0,Y 743.893,Z 762.06,A -85,B 0,C 180,E1 1573.023,E2 1573.023} C_VEL
LIN {X 0,Y 743.397,Z 762.06,A -85,B 0,C 180,E1 1577.887,E2 1577.887} C_VEL
LIN {X 0,Y 743.54,Z 762.06,A -85,B 0,C 180,E1 1582.43,E2 1582.43} C_VEL
LIN {X 0,Y 743.528,Z 762.06,A -85,B 0,C 180,E1 1586.733,E2 1586.733} C_VEL
LIN {X 0,Y 743.514,Z 762.06,A -85,B 0,C 180,E1 1590.92,E2 1590.92} C_VEL
LIN {X 0,Y 743.608,Z 762.06,A -85,B 0,C 180,E1 1594.75,E2 1594.75} C_VEL
LIN {X 0,Y 743.708,Z 762.06,A -85,B 0,C 180,E1 1599.803,E2 1599.803} C_VEL
LIN {X 0,Y 743.734,Z 762.06,A -85,B 0,C 180,E1 1605.897,E2 1605.897} C_VEL
LIN {X 0,Y 743.826,Z 762.06,A -85,B 0,C 180,E1 1610.655,E2 1610.655} C_VEL
LIN {X 0,Y 743.871,Z 762.06,A -85,B 0,C 180,E1 1614.504,E2 1614.504} C_VEL
LIN {X 0,Y 743.787,Z 762.06,A -85,B 0,C 180,E1 1618.843,E2 1618.843} C_VEL
LIN {X 0,Y 744.016,Z 762.06,A -85,B 0,C 180,E1 1620.929,E2 1620.929} C_VEL
LIN {X 0,Y 741.527,Z 762.06,A -85,B 0,C 180,E1 1621.92,E2 1621.92} C_VEL
LIN {X 0,Y 736.011,Z 762.06,A -85,B 0,C 180,E1 1623.398,E2 1623.398} C_VEL
LIN {X 0,Y 735.921,Z 762.06,A -85,B 0,C 180,E1 1623.569,E2 1623.569} C_VEL
LIN {X 0,Y 736.002,Z 762.06,A -85,B 0,C 180,E1 1628.269,E2 1628.269} C_VEL
LIN {X 0,Y 735.931,Z 762.06,A -85,B 0,C 180,E1 1633.059,E2 1633.059} C_VEL
LIN {X 0,Y 735.85,Z 762.06,A -85,B 0,C 180,E1 1637.946,E2 1637.946} C_VEL
LIN {X 0,Y 735.82,Z 762.06,A -85,B 0,C 180,E1 1642.46,E2 1642.46} C_VEL
LIN {X 0,Y 735.752,Z 762.06,A -85,B 0,C 180,E1 1646.866,E2 1646.866} C_VEL
LIN {X 0,Y 735.893,Z 762.06,A -85,B 0,C 180,E1 1652.272,E2 1652.272} C_VEL
LIN {X 0,Y 735.766,Z 762.06,A -85,B 0,C 180,E1 1656.775,E2 1656.775} C_VEL
LIN {X 0,Y 735.955,Z 762.06,A -85,B 0,C 180,E1 1662.657,E2 1662.657} C_VEL
LIN {X 0,Y 735.579,Z 762.06,A -85,B 0,C 180,E1 1667.318,E2 1667.318} C_VEL
LIN {X 0,Y 735.947,Z 762.292,A -85,B 0,C 180,E1 1672.087,E2 1672.087} C_VEL
LIN {X 0,Y 741.488,Z 773.897,A -85,B 0,C 180,E1 1672.559,E2 1672.559} C_VEL
LIN {X 0,Y 741.641,Z 847.049,A -85,B 0,C 180,E1 1673.547,E2 1673.547} C_VEL
LIN {X 0,Y 740.884,Z 891.436,A -85,B 0,C 180,E1 1674.559,E2 1674.559} C_VEL
LIN {X 0,Y 740.169,Z 939.21,A -85,B 0,C 180,E1 1676.173,E2 1676.173} C_VEL
LIN {X 0,Y 739.33,Z 986.808,A -85,B 0,C 180,E1 1678.342,E2 1678.342} C_VEL
LIN {X 0,Y 738.54,Z 1029.066,A -85,B 0,C 180,E1 1680.819,E2 1680.819} C_VEL
LIN {X 0,Y 737.766,Z 1068.747,A -85,B 0,C 180,E1 1683.695,E2 1683.695} C_VEL
LIN {X 0,Y 737.07,Z 1106.123,A -85,B 0,C 180,E1 1687.074,E2 1687.074} C_VEL
LIN {X 0,Y 736.608,Z 1136.485,A -85,B 0,C 180,E1 1690.488,E2 1690.488} C_VEL
LIN {X 0,Y 736.302,Z 1160.885,A -85,B 0,C 180,E1 1693.915,E2 1693.915} C_VEL
LIN {X 0,Y 736.192,Z 1179.72,A -85,B 0,C 180,E1 1697.285,E2 1697.285} C_VEL
LIN {X 0,Y 736.134,Z 1194.428,A -85,B 0,C 180,E1 1700.845,E2 1700.845} C_VEL
LIN {X 0,Y 736.009,Z 1204.631,A -85,B 0,C 180,E1 1704.611,E2 1704.611} C_VEL
LIN {X 0,Y 736.092,Z 1208.971,A -85,B 0,C 180,E1 1707.646,E2 1707.646} C_VEL
LIN {X 0,Y 736.231,Z 1209.669,A -85,B 0,C 180,E1 1711.175,E2 1711.175} C_VEL
LIN {X 0,Y 735.983,Z 1205.912,A -85,B 0,C 180,E1 1714.71,E2 1714.71} C_VEL
LIN {X 0,Y 735.952,Z 1197.335,A -85,B 0,C 180,E1 1718.263,E2 1718.263} C_VEL
LIN {X 0,Y 736.03,Z 1185.046,A -85,B 0,C 180,E1 1721.546,E2 1721.546} C_VEL
LIN {X 0,Y 736.216,Z 1167.347,A -85,B 0,C 180,E1 1725.017,E2 1725.017} C_VEL
LIN {X 0,Y 736.45,Z 1145.172,A -85,B 0,C 180,E1 1728.389,E2 1728.389} C_VEL
LIN {X 0,Y 736.907,Z 1116.959,A -85,B 0,C 180,E1 1731.789,E2 1731.789} C_VEL
LIN {X 0,Y 737.518,Z 1082.374,A -85,B 0,C 180,E1 1735.159,E2 1735.159} C_VEL
LIN {X 0,Y 738.295,Z 1041.535,A -85,B 0,C 180,E1 1738.344,E2 1738.344} C_VEL
LIN {X 0,Y 739.113,Z 1000.545,A -85,B 0,C 180,E1 1740.908,E2 1740.908} C_VEL
LIN {X 0,Y 740.021,Z 957.16,A -85,B 0,C 180,E1 1743.072,E2 1743.072} C_VEL
LIN {X 0,Y 740.778,Z 913.661,A -85,B 0,C 180,E1 1744.748,E2 1744.748} C_VEL
LIN {X 0,Y 741.301,Z 869.219,A -85,B 0,C 180,E1 1746.001,E2 1746.001} C_VEL
LIN {X 0,Y 741.675,Z 823.262,A -85,B 0,C 180,E1 1746.835,E2 1746.835} C_VEL
LIN {X 0,Y 741.061,Z 772.776,A -85,B 0,C 180,E1 1747.48,E2 1747.48} C_VEL
LIN {X 0,Y 735.987,Z 763.619,A -85,B 0,C 180,E1 1747.895,E2 1747.895} C_VEL
LIN {X 0,Y 735.833,Z 762.06,A -85,B 0,C 180,E1 1747.954,E2 1747.954} C_VEL
LIN {X 0,Y 735.94,Z 762.06,A -85,B 0,C 180,E1 1752.655,E2 1752.655} C_VEL
LIN {X 0,Y 735.576,Z 762.06,A -85,B 0,C 180,E1 1757.316,E2 1757.316} C_VEL
LIN {X 0,Y 735.632,Z 762.06,A -85,B 0,C 180,E1 1761.954,E2 1761.954} C_VEL
LIN {X 0,Y 735.669,Z 762.06,A -85,B 0,C 180,E1 1766.314,E2 1766.314} C_VEL
LIN {X 0,Y 735.674,Z 762.06,A -85,B 0,C 180,E1 1770.46,E2 1770.46} C_VEL
LIN {X 0,Y 735.797,Z 762.06,A -85,B 0,C 180,E1 1774.638,E2 1774.638} C_VEL
LIN {X 0,Y 735.741,Z 762.06,A -85,B 0,C 180,E1 1779.56,E2 1779.56} C_VEL
LIN {X 0,Y 735.916,Z 762.06,A -85,B 0,C 180,E1 1784.813,E2 1784.813} C_VEL
LIN {X 0,Y 735.823,Z 762.06,A -85,B 0,C 180,E1 1789.343,E2 1789.343} C_VEL
LIN {X 0,Y 735.878,Z 762.06,A -85,B 0,C 180,E1 1794.101,E2 1794.101} C_VEL
LIN {X 0,Y 736.154,Z 762.06,A -85,B 0,C 180,E1 1798.817,E2 1798.817} C_VEL
LIN {X 0,Y 736.046,Z 762.06,A -85,B 0,C 180,E1 1803.524,E2 1803.524} C_VEL
LIN {X 0,Y 735.83,Z 762.06,A -85,B 0,C 180,E1 1808.257,E2 1808.257} C_VEL
LIN {X 0,Y 735.739,Z 762.06,A -85,B 0,C 180,E1 1811.844,E2 1811.844} C_VEL
LIN {X 0,Y 735.621,Z 762.06,A -85,B 0,C 180,E1 1815.479,E2 1815.479} C_VEL
LIN {X 0,Y 735.809,Z 762.06,A -85,B 0,C 180,E1 1820.424,E2 1820.424} C_VEL
LIN {X 0,Y 735.675,Z 762.06,A -85,B 0,C 180,E1 1825.542,E2 1825.542} C_VEL
LIN {X 0,Y 735.635,Z 762.06,A -85,B 0,C 180,E1 1830.375,E2 1830.375} C_VEL
LIN {X 0,Y 735.659,Z 762.06,A -85,B 0,C 180,E1 1835.096,E2 1835.096} C_VEL
LIN {X 0,Y 735.498,Z 762.06,A -85,B 0,C 180,E1 1839.547,E2 1839.547} C_VEL
LIN {X 0,Y 735.51,Z 762.06,A -85,B 0,C 180,E1 1844.022,E2 1844.022} C_VEL
LIN {X 0,Y 736.017,Z 762.06,A -85,B 0,C 180,E1 1848.93,E2 1848.93} C_VEL
LIN {X 0,Y 735.95,Z 762.06,A -85,B 0,C 180,E1 1852.394,E2 1852.394} C_VEL
LIN {X 0,Y 740.718,Z 772.418,A -85,B 0,C 180,E1 1852.808,E2 1852.808} C_VEL
LIN {X 0,Y 741.702,Z 779.078,A -85,B 0,C 180,E1 1852.945,E2 1852.945} C_VEL
LIN {X 0,Y 741.513,Z 827.93,A -85,B 0,C 180,E1 1853.712,E2 1853.712} C_VEL
LIN {X 0,Y 740.79,Z 874.144,A -85,B 0,C 180,E1 1854.902,E2 1854.902} C_VEL
LIN {X 0,Y 740.083,Z 920.992,A -85,B 0,C 180,E1 1856.613,E2 1856.613} C_VEL
LIN {X 0,Y 739.217,Z 965.279,A -85,B 0,C 180,E1 1858.755,E2 1858.755} C_VEL
LIN {X 0,Y 738.359,Z 1008.904,A -85,B 0,C 180,E1 1861.425,E2 1861.425} C_VEL
LIN {X 0,Y 737.491,Z 1049.072,A -85,B 0,C 180,E1 1864.515,E2 1864.515} C_VEL
LIN {X 0,Y 736.954,Z 1082.358,A -85,B 0,C 180,E1 1867.673,E2 1867.673} C_VEL
LIN {X 0,Y 736.467,Z 1112.023,A -85,B 0,C 180,E1 1871.146,E2 1871.146} C_VEL
LIN {X 0,Y 736.259,Z 1134.964,A -85,B 0,C 180,E1 1874.526,E2 1874.526} C_VEL
LIN {X 0,Y 736.04,Z 1153.897,A -85,B 0,C 180,E1 1878.153,E2 1878.153} C_VEL
LIN {X 0,Y 736.092,Z 1165.6,A -85,B 0,C 180,E1 1881.144,E2 1881.144} C_VEL
LIN {X 0,Y 736.024,Z 1175.154,A -85,B 0,C 180,E1 1884.841,E2 1884.841} C_VEL
LIN {X 0,Y 735.984,Z 1179.012,A -85,B 0,C 180,E1 1887.647,E2 1887.647} C_VEL
LIN {X 0,Y 736.047,Z 1179.656,A -85,B 0,C 180,E1 1891.177,E2 1891.177} C_VEL
LIN {X 0,Y 736.191,Z 1175.013,A -85,B 0,C 180,E1 1895.141,E2 1895.141} C_VEL
LIN {X 0,Y 736.157,Z 1165.289,A -85,B 0,C 180,E1 1898.857,E2 1898.857} C_VEL
LIN {X 0,Y 736.245,Z 1150.976,A -85,B 0,C 180,E1 1902.404,E2 1902.404} C_VEL
LIN {X 0,Y 736.321,Z 1130.594,A -85,B 0,C 180,E1 1906.085,E2 1906.085} C_VEL
LIN {X 0,Y 736.63,Z 1104.607,A -85,B 0,C 180,E1 1909.707,E2 1909.707} C_VEL
LIN {X 0,Y 737.114,Z 1074.056,A -85,B 0,C 180,E1 1913.084,E2 1913.084} C_VEL
LIN {X 0,Y 737.823,Z 1037.937,A -85,B 0,C 180,E1 1916.321,E2 1916.321} C_VEL
LIN {X 0,Y 738.638,Z 996.083,A -85,B 0,C 180,E1 1919.331,E2 1919.331} C_VEL
LIN {X 0,Y 739.463,Z 954.078,A -85,B 0,C 180,E1 1921.746,E2 1921.746} C_VEL
LIN {X 0,Y 740.341,Z 908.642,A -85,B 0,C 180,E1 1923.797,E2 1923.797} C_VEL
LIN {X 0,Y 741.049,Z 863.028,A -85,B 0,C 180,E1 1925.341,E2 1925.341} C_VEL
LIN {X 0,Y 741.53,Z 818.444,A -85,B 0,C 180,E1 1926.388,E2 1926.388} C_VEL
LIN {X 0,Y 740.942,Z 772.482,A -85,B 0,C 180,E1 1927.088,E2 1927.088} C_VEL
LIN {X 0,Y 735.955,Z 762.06,A -85,B 0,C 180,E1 1927.575,E2 1927.575} C_VEL
LIN {X 0,Y 735.962,Z 762.06,A -85,B 0,C 180,E1 1932.655,E2 1932.655} C_VEL
LIN {X 0,Y 735.498,Z 762.06,A -85,B 0,C 180,E1 1937.701,E2 1937.701} C_VEL
LIN {X 0,Y 735.655,Z 762.06,A -85,B 0,C 180,E1 1941.973,E2 1941.973} C_VEL
LIN {X 0,Y 735.669,Z 762.06,A -85,B 0,C 180,E1 1946.33,E2 1946.33} C_VEL
LIN {X 0,Y 735.608,Z 762.06,A -85,B 0,C 180,E1 1950.473,E2 1950.473} C_VEL
LIN {X 0,Y 735.729,Z 762.06,A -85,B 0,C 180,E1 1954.652,E2 1954.652} C_VEL
LIN {X 0,Y 735.771,Z 762.06,A -85,B 0,C 180,E1 1959.575,E2 1959.575} C_VEL
LIN {X 0,Y 735.797,Z 762.06,A -85,B 0,C 180,E1 1965.742,E2 1965.742} C_VEL
LIN {X 0,Y 735.931,Z 762.06,A -85,B 0,C 180,E1 1970.553,E2 1970.553} C_VEL
LIN {X 0,Y 736.032,Z 762.06,A -85,B 0,C 180,E1 1974.116,E2 1974.116} C_VEL
LIN {X 0,Y 735.916,Z 762.06,A -85,B 0,C 180,E1 1978.83,E2 1978.83} C_VEL
LIN {X 0,Y 735.904,Z 762.06,A -85,B 0,C 180,E1 1982.36,E2 1982.36} C_VEL
LIN {X 0,Y 735.921,Z 762.06,A -85,B 0,C 180,E1 1983.569,E2 1983.569} C_VEL
LIN {X 0,Y 734.693,Z 762.06,A -85,B 0,C 180,E1 1984.243,E2 1984.243} C_VEL
LIN {X 0,Y 728.074,Z 762.06,A -85,B 0,C 180,E1 1986.074,E2 1986.074} C_VEL
LIN {X 0,Y 727.967,Z 762.06,A -85,B 0,C 180,E1 1986.248,E2 1986.248} C_VEL
LIN {X 0,Y 727.922,Z 762.06,A -85,B 0,C 180,E1 1990.774,E2 1990.774} C_VEL
LIN {X 0,Y 728.058,Z 762.06,A -85,B 0,C 180,E1 1995.659,E2 1995.659} C_VEL
LIN {X 0,Y 727.974,Z 762.06,A -85,B 0,C 180,E1 2000.915,E2 2000.915} C_VEL
LIN {X 0,Y 727.85,Z 762.06,A -85,B 0,C 180,E1 2005.852,E2 2005.852} C_VEL
LIN {X 0,Y 727.871,Z 762.06,A -85,B 0,C 180,E1 2009.889,E2 2009.889} C_VEL
LIN {X 0,Y 727.85,Z 762.06,A -85,B 0,C 180,E1 2014.098,E2 2014.098} C_VEL
LIN {X 0,Y 727.689,Z 762.06,A -85,B 0,C 180,E1 2018.537,E2 2018.537} C_VEL
LIN {X 0,Y 728.016,Z 762.06,A -85,B 0,C 180,E1 2023.407,E2 2023.407} C_VEL
LIN {X 0,Y 727.7,Z 762.06,A -85,B 0,C 180,E1 2028.382,E2 2028.382} C_VEL
LIN {X 0,Y 728.025,Z 762.201,A -85,B 0,C 180,E1 2031.599,E2 2031.599} C_VEL
LIN {X 0,Y 732.602,Z 772.141,A -85,B 0,C 180,E1 2032.003,E2 2032.003} C_VEL
LIN {X 0,Y 735.263,Z 778.527,A -85,B 0,C 180,E1 2032.242,E2 2032.242} C_VEL
LIN {X 0,Y 735.194,Z 849.377,A -85,B 0,C 180,E1 2033.22,E2 2033.22} C_VEL
LIN {X 0,Y 734.314,Z 895.445,A -85,B 0,C 180,E1 2034.31,E2 2034.31} C_VEL
LIN {X 0,Y 733.379,Z 943.659,A -85,B 0,C 180,E1 2036.004,E2 2036.004} C_VEL
LIN {X 0,Y 732.306,Z 989.731,A -85,B 0,C 180,E1 2038.157,E2 2038.157} C_VEL
LIN {X 0,Y 731.193,Z 1034.396,A -85,B 0,C 180,E1 2040.859,E2 2040.859} C_VEL
LIN {X 0,Y 730.258,Z 1072.277,A -85,B 0,C 180,E1 2043.706,E2 2043.706} C_VEL
LIN {X 0,Y 729.432,Z 1108.525,A -85,B 0,C 180,E1 2047.062,E2 2047.062} C_VEL
LIN {X 0,Y 728.799,Z 1139.226,A -85,B 0,C 180,E1 2050.624,E2 2050.624} C_VEL
LIN {X 0,Y 728.44,Z 1162.852,A -85,B 0,C 180,E1 2054.045,E2 2054.045} C_VEL
LIN {X 0,Y 728.223,Z 1181.85,A -85,B 0,C 180,E1 2057.609,E2 2057.609} C_VEL
LIN {X 0,Y 728.181,Z 1195.443,A -85,B 0,C 180,E1 2061.046,E2 2061.046} C_VEL
LIN {X 0,Y 728.178,Z 1203.568,A -85,B 0,C 180,E1 2064.044,E2 2064.044} C_VEL
LIN {X 0,Y 728.189,Z 1208.969,A -85,B 0,C 180,E1 2067.621,E2 2067.621} C_VEL
LIN {X 0,Y 728.329,Z 1209.669,A -85,B 0,C 180,E1 2071.188,E2 2071.188} C_VEL
LIN {X 0,Y 728.096,Z 1205.478,A -85,B 0,C 180,E1 2074.997,E2 2074.997} C_VEL
LIN {X 0,Y 728.064,Z 1197.335,A -85,B 0,C 180,E1 2078.353,E2 2078.353} C_VEL
LIN {X 0,Y 728.158,Z 1185.047,A -85,B 0,C 180,E1 2081.673,E2 2081.673} C_VEL
LIN {X 0,Y 728.383,Z 1167.775,A -85,B 0,C 180,E1 2085.108,E2 2085.108} C_VEL
LIN {X 0,Y 728.691,Z 1145.174,A -85,B 0,C 180,E1 2088.592,E2 2088.592} C_VEL
LIN {X 0,Y 729.205,Z 1117.094,A -85,B 0,C 180,E1 2092.016,E2 2092.016} C_VEL
LIN {X 0,Y 730.042,Z 1082.373,A -85,B 0,C 180,E1 2095.435,E2 2095.435} C_VEL
LIN {X 0,Y 731.013,Z 1041.534,A -85,B 0,C 180,E1 2098.652,E2 2098.652} C_VEL
LIN {X 0,Y 732.053,Z 1000.232,A -85,B 0,C 180,E1 2101.257,E2 2101.257} C_VEL
LIN {X 0,Y 733.216,Z 956.448,A -85,B 0,C 180,E1 2103.452,E2 2103.452} C_VEL
LIN {X 0,Y 734.133,Z 913.051,A -85,B 0,C 180,E1 2105.128,E2 2105.128} C_VEL
LIN {X 0,Y 734.884,Z 868.233,A -85,B 0,C 180,E1 2106.389,E2 2106.389} C_VEL
LIN {X 0,Y 735.342,Z 823.235,A -85,B 0,C 180,E1 2107.205,E2 2107.205} C_VEL
LIN {X 0,Y 734.579,Z 775.827,A -85,B 0,C 180,E1 2107.832,E2 2107.832} C_VEL
LIN {X 0,Y 727.772,Z 762.06,A -85,B 0,C 180,E1 2108.448,E2 2108.448} C_VEL
LIN {X 0,Y 728.019,Z 762.06,A -85,B 0,C 180,E1 2113.406,E2 2113.406} C_VEL
LIN {X 0,Y 727.694,Z 762.06,A -85,B 0,C 180,E1 2118.379,E2 2118.379} C_VEL
LIN {X 0,Y 727.688,Z 762.06,A -85,B 0,C 180,E1 2122.968,E2 2122.968} C_VEL
LIN {X 0,Y 727.701,Z 762.06,A -85,B 0,C 180,E1 2127.319,E2 2127.319} C_VEL
LIN {X 0,Y 727.668,Z 762.06,A -85,B 0,C 180,E1 2131.465,E2 2131.465} C_VEL
LIN {X 0,Y 727.744,Z 762.06,A -85,B 0,C 180,E1 2136.01,E2 2136.01} C_VEL
LIN {X 0,Y 727.775,Z 762.06,A -85,B 0,C 180,E1 2140.592,E2 2140.592} C_VEL
LIN {X 0,Y 728.049,Z 762.06,A -85,B 0,C 180,E1 2144.341,E2 2144.341} C_VEL
LIN {X 0,Y 727.919,Z 762.06,A -85,B 0,C 180,E1 2149.226,E2 2149.226} C_VEL
LIN {X 0,Y 727.996,Z 762.06,A -85,B 0,C 180,E1 2154.037,E2 2154.037} C_VEL
LIN {X 0,Y 728.248,Z 762.06,A -85,B 0,C 180,E1 2158.804,E2 2158.804} C_VEL
LIN {X 0,Y 728.137,Z 762.06,A -85,B 0,C 180,E1 2163.562,E2 2163.562} C_VEL
LIN {X 0,Y 727.94,Z 762.06,A -85,B 0,C 180,E1 2168.347,E2 2168.347} C_VEL
LIN {X 0,Y 727.81,Z 762.06,A -85,B 0,C 180,E1 2172.625,E2 2172.625} C_VEL
LIN {X 0,Y 727.49,Z 762.06,A -85,B 0,C 180,E1 2177.161,E2 2177.161} C_VEL
LIN {X 0,Y 727.757,Z 762.06,A -85,B 0,C 180,E1 2181.937,E2 2181.937} C_VEL
LIN {X 0,Y 727.738,Z 762.06,A -85,B 0,C 180,E1 2186.765,E2 2186.765} C_VEL
LIN {X 0,Y 727.797,Z 762.06,A -85,B 0,C 180,E1 2191.651,E2 2191.651} C_VEL
LIN {X 0,Y 727.845,Z 762.06,A -85,B 0,C 180,E1 2197.005,E2 2197.005} C_VEL
LIN {X 0,Y 727.743,Z 762.06,A -85,B 0,C 180,E1 2201.625,E2 2201.625} C_VEL
LIN {X 0,Y 727.806,Z 762.06,A -85,B 0,C 180,E1 2206.752,E2 2206.752} C_VEL
LIN {X 0,Y 728.002,Z 762.06,A -85,B 0,C 180,E1 2211.487,E2 2211.487} C_VEL
LIN {X 0,Y 728.046,Z 762.803,A -85,B 0,C 180,E1 2211.931,E2 2211.931} C_VEL
LIN {X 0,Y 735.391,Z 777.435,A -85,B 0,C 180,E1 2212.554,E2 2212.554} C_VEL
LIN {X 0,Y 735.075,Z 826.787,A -85,B 0,C 180,E1 2213.317,E2 2213.317} C_VEL
LIN {X 0,Y 734.19,Z 874.129,A -85,B 0,C 180,E1 2214.539,E2 2214.539} C_VEL
LIN {X 0,Y 733.321,Z 921.049,A -85,B 0,C 180,E1 2216.267,E2 2216.267} C_VEL
LIN {X 0,Y 732.21,Z 965.126,A -85,B 0,C 180,E1 2218.414,E2 2218.414} C_VEL
LIN {X 0,Y 731.102,Z 1009.135,A -85,B 0,C 180,E1 2221.131,E2 2221.131} C_VEL
LIN {X 0,Y 729.993,Z 1049.065,A -85,B 0,C 180,E1 2224.234,E2 2224.234} C_VEL
LIN {X 0,Y 729.308,Z 1081.894,A -85,B 0,C 180,E1 2227.376,E2 2227.376} C_VEL
LIN {X 0,Y 728.725,Z 1112.021,A -85,B 0,C 180,E1 2230.938,E2 2230.938} C_VEL
LIN {X 0,Y 728.461,Z 1134.963,A -85,B 0,C 180,E1 2234.356,E2 2234.356} C_VEL
LIN {X 0,Y 728.174,Z 1153.896,A -85,B 0,C 180,E1 2238.024,E2 2238.024} C_VEL
LIN {X 0,Y 728.226,Z 1165.599,A -85,B 0,C 180,E1 2241.047,E2 2241.047} C_VEL
LIN {X 0,Y 728.128,Z 1175.217,A -85,B 0,C 180,E1 2244.82,E2 2244.82} C_VEL
LIN {X 0,Y 728.08,Z 1179.009,A -85,B 0,C 180,E1 2247.622,E2 2247.622} C_VEL
LIN {X 0,Y 728.145,Z 1179.656,A -85,B 0,C 180,E1 2251.19,E2 2251.19} C_VEL
LIN {X 0,Y 728.335,Z 1175.832,A -85,B 0,C 180,E1 2254.761,E2 2254.761} C_VEL
LIN {X 0,Y 728.316,Z 1167.193,A -85,B 0,C 180,E1 2258.352,E2 2258.352} C_VEL
LIN {X 0,Y 728.363,Z 1153.49,A -85,B 0,C 180,E1 2261.975,E2 2261.975} C_VEL
LIN {X 0,Y 728.539,Z 1134.443,A -85,B 0,C 180,E1 2265.644,E2 2265.644} C_VEL
LIN {X 0,Y 728.936,Z 1108.878,A -85,B 0,C 180,E1 2269.372,E2 2269.372} C_VEL
LIN {X 0,Y 729.44,Z 1078.786,A -85,B 0,C 180,E1 2272.866,E2 2272.866} C_VEL
LIN {X 0,Y 730.304,Z 1041.615,A -85,B 0,C 180,E1 2276.305,E2 2276.305} C_VEL
LIN {X 0,Y 731.206,Z 1003.732,A -85,B 0,C 180,E1 2279.14,E2 2279.14} C_VEL
LIN {X 0,Y 732.359,Z 960.09,A -85,B 0,C 180,E1 2281.775,E2 2281.775} C_VEL
LIN {X 0,Y 733.415,Z 915.515,A -85,B 0,C 180,E1 2283.871,E2 2283.871} C_VEL
LIN {X 0,Y 734.33,Z 869.049,A -85,B 0,C 180,E1 2285.529,E2 2285.529} C_VEL
LIN {X 0,Y 735.082,Z 821.057,A -85,B 0,C 180,E1 2286.708,E2 2286.708} C_VEL
LIN {X 0,Y 734.645,Z 775.796,A -85,B 0,C 180,E1 2287.42,E2 2287.42} C_VEL
LIN {X 0,Y 727.889,Z 762.06,A -85,B 0,C 180,E1 2288.033,E2 2288.033} C_VEL
LIN {X 0,Y 727.997,Z 762.06,A -85,B 0,C 180,E1 2293.424,E2 2293.424} C_VEL
LIN {X 0,Y 727.651,Z 762.06,A -85,B 0,C 180,E1 2298.385,E2 2298.385} C_VEL
LIN {X 0,Y 727.728,Z 762.06,A -85,B 0,C 180,E1 2302.988,E2 2302.988} C_VEL
LIN {X 0,Y 727.697,Z 762.06,A -85,B 0,C 180,E1 2307.336,E2 2307.336} C_VEL
LIN {X 0,Y 727.61,Z 762.06,A -85,B 0,C 180,E1 2311.479,E2 2311.479} C_VEL
LIN {X 0,Y 727.564,Z 762.06,A -85,B 0,C 180,E1 2316.045,E2 2316.045} C_VEL
LIN {X 0,Y 727.755,Z 762.06,A -85,B 0,C 180,E1 2320.606,E2 2320.606} C_VEL
LIN {X 0,Y 727.883,Z 762.06,A -85,B 0,C 180,E1 2325.583,E2 2325.583} C_VEL
LIN {X 0,Y 728.049,Z 762.06,A -85,B 0,C 180,E1 2330.45,E2 2330.45} C_VEL
LIN {X 0,Y 727.993,Z 762.06,A -85,B 0,C 180,E1 2335.245,E2 2335.245} C_VEL
LIN {X 0,Y 728.102,Z 762.06,A -85,B 0,C 180,E1 2340.007,E2 2340.007} C_VEL
LIN {X 0,Y 728.142,Z 762.06,A -85,B 0,C 180,E1 2345.028,E2 2345.028} C_VEL
LIN {X 0,Y 727.967,Z 762.06,A -85,B 0,C 180,E1 2346.248,E2 2346.248} C_VEL
LIN {X 0,Y 724.034,Z 762.06,A -85,B 0,C 180,E1 2347.589,E2 2347.589} C_VEL
LIN {X 0,Y 720.108,Z 762.06,A -85,B 0,C 180,E1 2348.946,E2 2348.946} C_VEL
LIN {X 0,Y 720.072,Z 762.06,A -85,B 0,C 180,E1 2353.352,E2 2353.352} C_VEL
LIN {X 0,Y 720.059,Z 762.06,A -85,B 0,C 180,E1 2358.353,E2 2358.353} C_VEL
LIN {X 0,Y 720.064,Z 762.06,A -85,B 0,C 180,E1 2363.503,E2 2363.503} C_VEL
LIN {X 0,Y 719.984,Z 762.06,A -85,B 0,C 180,E1 2368.868,E2 2368.868} C_VEL
LIN {X 0,Y 720.013,Z 762.06,A -85,B 0,C 180,E1 2373.074,E2 2373.074} C_VEL
LIN {X 0,Y 719.909,Z 762.06,A -85,B 0,C 180,E1 2377.5,E2 2377.5} C_VEL
LIN {X 0,Y 720.019,Z 762.06,A -85,B 0,C 180,E1 2382.73,E2 2382.73} C_VEL
LIN {X 0,Y 719.761,Z 762.06,A -85,B 0,C 180,E1 2387.294,E2 2387.294} C_VEL
LIN {X 0,Y 720.097,Z 762.706,A -85,B 0,C 180,E1 2391.103,E2 2391.103} C_VEL
LIN {X 0,Y 729.038,Z 781.138,A -85,B 0,C 180,E1 2391.894,E2 2391.894} C_VEL
LIN {X 0,Y 728.861,Z 849.482,A -85,B 0,C 180,E1 2392.849,E2 2392.849} C_VEL
LIN {X 0,Y 727.814,Z 894.637,A -85,B 0,C 180,E1 2393.918,E2 2393.918} C_VEL
LIN {X 0,Y 726.628,Z 942.134,A -85,B 0,C 180,E1 2395.579,E2 2395.579} C_VEL
LIN {X 0,Y 725.351,Z 989.498,A -85,B 0,C 180,E1 2397.802,E2 2397.802} C_VEL
LIN {X 0,Y 724.027,Z 1033.402,A -85,B 0,C 180,E1 2400.474,E2 2400.474} C_VEL
LIN {X 0,Y 722.88,Z 1070.957,A -85,B 0,C 180,E1 2403.301,E2 2403.301} C_VEL
LIN {X 0,Y 721.868,Z 1107.743,A -85,B 0,C 180,E1 2406.728,E2 2406.728} C_VEL
LIN {X 0,Y 721.129,Z 1138.01,A -85,B 0,C 180,E1 2410.251,E2 2410.251} C_VEL
LIN {X 0,Y 720.66,Z 1162.85,A -85,B 0,C 180,E1 2413.869,E2 2413.869} C_VEL
LIN {X 0,Y 720.39,Z 1181.879,A -85,B 0,C 180,E1 2417.478,E2 2417.478} C_VEL
LIN {X 0,Y 720.343,Z 1195.443,A -85,B 0,C 180,E1 2420.947,E2 2420.947} C_VEL
LIN {X 0,Y 720.212,Z 1204.797,A -85,B 0,C 180,E1 2424.582,E2 2424.582} C_VEL
LIN {X 0,Y 720.286,Z 1208.966,A -85,B 0,C 180,E1 2427.595,E2 2427.595} C_VEL
LIN {X 0,Y 720.44,Z 1209.669,A -85,B 0,C 180,E1 2431.201,E2 2431.201} C_VEL
LIN {X 0,Y 720.215,Z 1205.912,A -85,B 0,C 180,E1 2434.814,E2 2434.814} C_VEL
LIN {X 0,Y 720.174,Z 1197.334,A -85,B 0,C 180,E1 2438.445,E2 2438.445} C_VEL
LIN {X 0,Y 720.288,Z 1185.048,A -85,B 0,C 180,E1 2441.802,E2 2441.802} C_VEL
LIN {X 0,Y 720.539,Z 1167.83,A -85,B 0,C 180,E1 2445.267,E2 2445.267} C_VEL
LIN {X 0,Y 720.887,Z 1146.561,A -85,B 0,C 180,E1 2448.601,E2 2448.601} C_VEL
LIN {X 0,Y 721.572,Z 1119.839,A -85,B 0,C 180,E1 2451.959,E2 2451.959} C_VEL
LIN {X 0,Y 722.475,Z 1084.899,A -85,B 0,C 180,E1 2455.487,E2 2455.487} C_VEL
LIN {X 0,Y 723.56,Z 1047.069,A -85,B 0,C 180,E1 2458.562,E2 2458.562} C_VEL
LIN {X 0,Y 724.934,Z 1005.089,A -85,B 0,C 180,E1 2461.319,E2 2461.319} C_VEL
LIN {X 0,Y 726.259,Z 961.551,A -85,B 0,C 180,E1 2463.572,E2 2463.572} C_VEL
LIN {X 0,Y 727.466,Z 917.496,A -85,B 0,C 180,E1 2465.342,E2 2465.342} C_VEL
LIN {X 0,Y 728.391,Z 871.754,A -85,B 0,C 180,E1 2466.68,E2 2466.68} C_VEL
LIN {X 0,Y 729.026,Z 825.025,A -85,B 0,C 180,E1 2467.557,E2 2467.557} C_VEL
LIN {X 0,Y 728.438,Z 779.06,A -85,B 0,C 180,E1 2468.168,E2 2468.168} C_VEL
LIN {X 0,Y 719.813,Z 762.82,A -85,B 0,C 180,E1 2468.914,E2 2468.914} C_VEL
LIN {X 0,Y 720.074,Z 762.06,A -85,B 0,C 180,E1 2473.829,E2 2473.829} C_VEL
LIN {X 0,Y 719.869,Z 762.06,A -85,B 0,C 180,E1 2479.4,E2 2479.4} C_VEL
LIN {X 0,Y 719.82,Z 762.06,A -85,B 0,C 180,E1 2484.956,E2 2484.956} C_VEL
LIN {X 0,Y 719.887,Z 762.06,A -85,B 0,C 180,E1 2489.746,E2 2489.746} C_VEL
LIN {X 0,Y 719.871,Z 762.06,A -85,B 0,C 180,E1 2495.172,E2 2495.172} C_VEL
LIN {X 0,Y 719.866,Z 762.06,A -85,B 0,C 180,E1 2500.37,E2 2500.37} C_VEL
LIN {X 0,Y 720.07,Z 762.06,A -85,B 0,C 180,E1 2504.868,E2 2504.868} C_VEL
LIN {X 0,Y 720.036,Z 762.06,A -85,B 0,C 180,E1 2509.107,E2 2509.107} C_VEL
LIN {X 0,Y 720.086,Z 762.06,A -85,B 0,C 180,E1 2513.971,E2 2513.971} C_VEL
LIN {X 0,Y 720.359,Z 762.06,A -85,B 0,C 180,E1 2518.791,E2 2518.791} C_VEL
LIN {X 0,Y 720.252,Z 762.06,A -85,B 0,C 180,E1 2523.601,E2 2523.601} C_VEL
LIN {X 0,Y 720.037,Z 762.06,A -85,B 0,C 180,E1 2528.44,E2 2528.44} C_VEL
LIN {X 0,Y 719.924,Z 762.06,A -85,B 0,C 180,E1 2532.108,E2 2532.108} C_VEL
LIN {X 0,Y 719.741,Z 762.06,A -85,B 0,C 180,E1 2535.83,E2 2535.83} C_VEL
LIN {X 0,Y 719.94,Z 762.06,A -85,B 0,C 180,E1 2540.895,E2 2540.895} C_VEL
LIN {X 0,Y 719.826,Z 762.06,A -85,B 0,C 180,E1 2546.147,E2 2546.147} C_VEL
LIN {X 0,Y 719.817,Z 762.06,A -85,B 0,C 180,E1 2550.605,E2 2550.605} C_VEL
LIN {X 0,Y 719.812,Z 762.06,A -85,B 0,C 180,E1 2555.043,E2 2555.043} C_VEL
LIN {X 0,Y 719.728,Z 762.06,A -85,B 0,C 180,E1 2559.029,E2 2559.029} C_VEL
LIN {X 0,Y 719.67,Z 762.06,A -85,B 0,C 180,E1 2563.844,E2 2563.844} C_VEL
LIN {X 0,Y 720.124,Z 762.06,A -85,B 0,C 180,E1 2569.421,E2 2569.421} C_VEL
LIN {X 0,Y 720.145,Z 762.684,A -85,B 0,C 180,E1 2571.437,E2 2571.437} C_VEL
LIN {X 0,Y 729.108,Z 780.583,A -85,B 0,C 180,E1 2572.214,E2 2572.214} C_VEL
LIN {X 0,Y 728.69,Z 828.736,A -85,B 0,C 180,E1 2572.987,E2 2572.987} C_VEL
LIN {X 0,Y 727.606,Z 876.029,A -85,B 0,C 180,E1 2574.232,E2 2574.232} C_VEL
LIN {X 0,Y 726.532,Z 922.697,A -85,B 0,C 180,E1 2575.979,E2 2575.979} C_VEL
LIN {X 0,Y 725.12,Z 967.682,A -85,B 0,C 180,E1 2578.217,E2 2578.217} C_VEL
LIN {X 0,Y 723.853,Z 1010.011,A -85,B 0,C 180,E1 2580.879,E2 2580.879} C_VEL
LIN {X 0,Y 722.519,Z 1050.104,A -85,B 0,C 180,E1 2584.038,E2 2584.038} C_VEL
LIN {X 0,Y 721.626,Z 1083.703,A -85,B 0,C 180,E1 2587.322,E2 2587.322} C_VEL
LIN {X 0,Y 720.968,Z 1112.753,A -85,B 0,C 180,E1 2590.823,E2 2590.823} C_VEL
LIN {X 0,Y 720.653,Z 1134.961,A -85,B 0,C 180,E1 2594.182,E2 2594.182} C_VEL
LIN {X 0,Y 720.341,Z 1153.895,A -85,B 0,C 180,E1 2597.891,E2 2597.891} C_VEL
LIN {X 0,Y 720.24,Z 1167.471,A -85,B 0,C 180,E1 2601.555,E2 2601.555} C_VEL
LIN {X 0,Y 720.178,Z 1175.982,A -85,B 0,C 180,E1 2605.186,E2 2605.186} C_VEL
LIN {X 0,Y 720.127,Z 1179.682,A -85,B 0,C 180,E1 2608.798,E2 2608.798} C_VEL
LIN {X 0,Y 720.154,Z 1178.927,A -85,B 0,C 180,E1 2612.406,E2 2612.406} C_VEL
LIN {X 0,Y 720.215,Z 1173.471,A -85,B 0,C 180,E1 2616.022,E2 2616.022} C_VEL
LIN {X 0,Y 720.264,Z 1163.26,A -85,B 0,C 180,E1 2619.663,E2 2619.663} C_VEL
LIN {X 0,Y 720.421,Z 1147.782,A -85,B 0,C 180,E1 2623.341,E2 2623.341} C_VEL
LIN {X 0,Y 720.692,Z 1128.631,A -85,B 0,C 180,E1 2626.757,E2 2626.757} C_VEL
LIN {X 0,Y 721.254,Z 1102.77,A -85,B 0,C 180,E1 2630.385,E2 2630.385} C_VEL
LIN {X 0,Y 721.996,Z 1070.335,A -85,B 0,C 180,E1 2633.976,E2 2633.976} C_VEL
LIN {X 0,Y 723,Z 1035.223,A -85,B 0,C 180,E1 2637.123,E2 2637.123} C_VEL
LIN {X 0,Y 724.315,Z 994.968,A -85,B 0,C 180,E1 2640.047,E2 2640.047} C_VEL
LIN {X 0,Y 725.641,Z 952.16,A -85,B 0,C 180,E1 2642.526,E2 2642.526} C_VEL
LIN {X 0,Y 727.005,Z 907.216,A -85,B 0,C 180,E1 2644.565,E2 2644.565} C_VEL
LIN {X 0,Y 728.053,Z 863.036,A -85,B 0,C 180,E1 2646.071,E2 2646.071} C_VEL
LIN {X 0,Y 728.825,Z 817.726,A -85,B 0,C 180,E1 2647.142,E2 2647.142} C_VEL
LIN {X 0,Y 728.468,Z 778.936,A -85,B 0,C 180,E1 2647.755,E2 2647.755} C_VEL
LIN {X 0,Y 720.069,Z 763.687,A -85,B 0,C 180,E1 2648.466,E2 2648.466} C_VEL
LIN {X 0,Y 719.873,Z 762.06,A -85,B 0,C 180,E1 2648.575,E2 2648.575} C_VEL
LIN {X 0,Y 720.059,Z 762.06,A -85,B 0,C 180,E1 2653.832,E2 2653.832} C_VEL
LIN {X 0,Y 719.836,Z 762.06,A -85,B 0,C 180,E1 2659.416,E2 2659.416} C_VEL
LIN {X 0,Y 719.837,Z 762.06,A -85,B 0,C 180,E1 2664.014,E2 2664.014} C_VEL
LIN {X 0,Y 719.806,Z 762.06,A -85,B 0,C 180,E1 2669.399,E2 2669.399} C_VEL
LIN {X 0,Y 719.841,Z 762.06,A -85,B 0,C 180,E1 2674.512,E2 2674.512} C_VEL
LIN {X 0,Y 719.845,Z 762.06,A -85,B 0,C 180,E1 2680.384,E2 2680.384} C_VEL
LIN {X 0,Y 719.938,Z 762.06,A -85,B 0,C 180,E1 2685.421,E2 2685.421} C_VEL
LIN {X 0,Y 720.145,Z 762.06,A -85,B 0,C 180,E1 2690.481,E2 2690.481} C_VEL
LIN {X 0,Y 720.111,Z 762.06,A -85,B 0,C 180,E1 2695.193,E2 2695.193} C_VEL
LIN {X 0,Y 720.22,Z 762.06,A -85,B 0,C 180,E1 2700.007,E2 2700.007} C_VEL
LIN {X 0,Y 720.303,Z 762.06,A -85,B 0,C 180,E1 2704.82,E2 2704.82} C_VEL
LIN {X 0,Y 720.108,Z 762.06,A -85,B 0,C 180,E1 2708.946,E2 2708.946} C_VEL
LIN {X 0,Y 716.078,Z 762.06,A -85,B 0,C 180,E1 2710.301,E2 2710.301} C_VEL
LIN {X 0,Y 712.125,Z 762.06,A -85,B 0,C 180,E1 2711.671,E2 2711.671} C_VEL
LIN {X 0,Y 712.256,Z 762.06,A -85,B 0,C 180,E1 2717.307,E2 2717.307} C_VEL
LIN {X 0,Y 712.093,Z 762.06,A -85,B 0,C 180,E1 2722.461,E2 2722.461} C_VEL
LIN {X 0,Y 712.009,Z 762.06,A -85,B 0,C 180,E1 2726.952,E2 2726.952} C_VEL
LIN {X 0,Y 712.061,Z 762.06,A -85,B 0,C 180,E1 2732.046,E2 2732.046} C_VEL
LIN {X 0,Y 711.991,Z 762.06,A -85,B 0,C 180,E1 2736.464,E2 2736.464} C_VEL
LIN {X 0,Y 712.032,Z 762.06,A -85,B 0,C 180,E1 2742.03,E2 2742.03} C_VEL
LIN {X 0,Y 711.962,Z 762.06,A -85,B 0,C 180,E1 2746.192,E2 2746.192} C_VEL
LIN {X 0,Y 712.092,Z 762.219,A -85,B 0,C 180,E1 2750.575,E2 2750.575} C_VEL
LIN {X 0,Y 717.058,Z 772.576,A -85,B 0,C 180,E1 2751.032,E2 2751.032} C_VEL
LIN {X 0,Y 722.807,Z 783.043,A -85,B 0,C 180,E1 2751.53,E2 2751.53} C_VEL
LIN {X 0,Y 722.532,Z 849.84,A -85,B 0,C 180,E1 2752.475,E2 2752.475} C_VEL
LIN {X 0,Y 721.304,Z 895.802,A -85,B 0,C 180,E1 2753.575,E2 2753.575} C_VEL
LIN {X 0,Y 719.881,Z 945.098,A -85,B 0,C 180,E1 2755.338,E2 2755.338} C_VEL
LIN {X 0,Y 718.372,Z 989.809,A -85,B 0,C 180,E1 2757.469,E2 2757.469} C_VEL
LIN {X 0,Y 716.826,Z 1033.44,A -85,B 0,C 180,E1 2760.15,E2 2760.15} C_VEL
LIN {X 0,Y 715.446,Z 1071.671,A -85,B 0,C 180,E1 2763.064,E2 2763.064} C_VEL
LIN {X 0,Y 714.341,Z 1107.74,A -85,B 0,C 180,E1 2766.468,E2 2766.468} C_VEL
LIN {X 0,Y 713.387,Z 1138.012,A -85,B 0,C 180,E1 2770.027,E2 2770.027} C_VEL
LIN {X 0,Y 712.848,Z 1162.849,A -85,B 0,C 180,E1 2773.687,E2 2773.687} C_VEL
LIN {X 0,Y 712.543,Z 1181.716,A -85,B 0,C 180,E1 2777.3,E2 2777.3} C_VEL
LIN {X 0,Y 712.476,Z 1195.664,A -85,B 0,C 180,E1 2780.916,E2 2780.916} C_VEL
LIN {X 0,Y 712.328,Z 1204.797,A -85,B 0,C 180,E1 2784.522,E2 2784.522} C_VEL
LIN {X 0,Y 712.383,Z 1208.963,A -85,B 0,C 180,E1 2787.568,E2 2787.568} C_VEL
LIN {X 0,Y 712.537,Z 1209.669,A -85,B 0,C 180,E1 2791.215,E2 2791.215} C_VEL
LIN {X 0,Y 712.333,Z 1205.912,A -85,B 0,C 180,E1 2794.867,E2 2794.867} C_VEL
LIN {X 0,Y 712.291,Z 1197.334,A -85,B 0,C 180,E1 2798.54,E2 2798.54} C_VEL
LIN {X 0,Y 712.402,Z 1185.049,A -85,B 0,C 180,E1 2801.935,E2 2801.935} C_VEL
LIN {X 0,Y 712.706,Z 1167.832,A -85,B 0,C 180,E1 2805.439,E2 2805.439} C_VEL
LIN {X 0,Y 713.114,Z 1146.743,A -85,B 0,C 180,E1 2808.785,E2 2808.785} C_VEL
LIN {X 0,Y 713.87,Z 1119.476,A -85,B 0,C 180,E1 2812.249,E2 2812.249} C_VEL
LIN {X 0,Y 715.009,Z 1084.29,A -85,B 0,C 180,E1 2815.831,E2 2815.831} C_VEL
LIN {X 0,Y 716.325,Z 1047.07,A -85,B 0,C 180,E1 2818.878,E2 2818.878} C_VEL
LIN {X 0,Y 717.901,Z 1005.85,A -85,B 0,C 180,E1 2821.617,E2 2821.617} C_VEL
LIN {X 0,Y 719.444,Z 962.642,A -85,B 0,C 180,E1 2823.881,E2 2823.881} C_VEL
LIN {X 0,Y 720.849,Z 919.004,A -85,B 0,C 180,E1 2825.658,E2 2825.658} C_VEL
LIN {X 0,Y 721.977,Z 873.203,A -85,B 0,C 180,E1 2827.023,E2 2827.023} C_VEL
LIN {X 0,Y 722.732,Z 826.531,A -85,B 0,C 180,E1 2827.919,E2 2827.919} C_VEL
LIN {X 0,Y 722.328,Z 782.373,A -85,B 0,C 180,E1 2828.509,E2 2828.509} C_VEL
LIN {X 0,Y 712.008,Z 763.76,A -85,B 0,C 180,E1 2829.41,E2 2829.41} C_VEL
LIN {X 0,Y 711.805,Z 762.06,A -85,B 0,C 180,E1 2829.559,E2 2829.559} C_VEL
LIN {X 0,Y 712.175,Z 762.06,A -85,B 0,C 180,E1 2834.442,E2 2834.442} C_VEL
LIN {X 0,Y 711.97,Z 762.06,A -85,B 0,C 180,E1 2840.448,E2 2840.448} C_VEL
LIN {X 0,Y 711.881,Z 762.06,A -85,B 0,C 180,E1 2845.878,E2 2845.878} C_VEL
LIN {X 0,Y 711.877,Z 762.06,A -85,B 0,C 180,E1 2850.772,E2 2850.772} C_VEL
LIN {X 0,Y 711.922,Z 762.06,A -85,B 0,C 180,E1 2855.881,E2 2855.881} C_VEL
LIN {X 0,Y 711.948,Z 762.06,A -85,B 0,C 180,E1 2860.143,E2 2860.143} C_VEL
LIN {X 0,Y 712.219,Z 762.06,A -85,B 0,C 180,E1 2863.984,E2 2863.984} C_VEL
LIN {X 0,Y 712.129,Z 762.06,A -85,B 0,C 180,E1 2868.984,E2 2868.984} C_VEL
LIN {X 0,Y 712.177,Z 762.06,A -85,B 0,C 180,E1 2873.904,E2 2873.904} C_VEL
LIN {X 0,Y 712.452,Z 762.06,A -85,B 0,C 180,E1 2878.778,E2 2878.778} C_VEL
LIN {X 0,Y 712.343,Z 762.06,A -85,B 0,C 180,E1 2883.641,E2 2883.641} C_VEL
LIN {X 0,Y 712.136,Z 762.06,A -85,B 0,C 180,E1 2888.534,E2 2888.534} C_VEL
LIN {X 0,Y 711.992,Z 762.06,A -85,B 0,C 180,E1 2892.504,E2 2892.504} C_VEL
LIN {X 0,Y 711.687,Z 762.06,A -85,B 0,C 180,E1 2897.283,E2 2897.283} C_VEL
LIN {X 0,Y 712.019,Z 762.06,A -85,B 0,C 180,E1 2901.138,E2 2901.138} C_VEL
LIN {X 0,Y 711.893,Z 762.06,A -85,B 0,C 180,E1 2906.46,E2 2906.46} C_VEL
LIN {X 0,Y 711.982,Z 762.06,A -85,B 0,C 180,E1 2911.902,E2 2911.902} C_VEL
LIN {X 0,Y 711.979,Z 762.06,A -85,B 0,C 180,E1 2916.447,E2 2916.447} C_VEL
LIN {X 0,Y 711.851,Z 762.06,A -85,B 0,C 180,E1 2922.015,E2 2922.015} C_VEL
LIN {X 0,Y 712.122,Z 762.06,A -85,B 0,C 180,E1 2927.943,E2 2927.943} C_VEL
LIN {X 0,Y 712.266,Z 762.757,A -85,B 0,C 180,E1 2930.931,E2 2930.931} C_VEL
LIN {X 0,Y 722.856,Z 783.424,A -85,B 0,C 180,E1 2931.864,E2 2931.864} C_VEL
LIN {X 0,Y 722.296,Z 830.685,A -85,B 0,C 180,E1 2932.649,E2 2932.649} C_VEL
LIN {X 0,Y 721.061,Z 876.639,A -85,B 0,C 180,E1 2933.878,E2 2933.878} C_VEL
LIN {X 0,Y 719.785,Z 922.189,A -85,B 0,C 180,E1 2935.595,E2 2935.595} C_VEL
LIN {X 0,Y 718.158,Z 966.668,A -85,B 0,C 180,E1 2937.813,E2 2937.813} C_VEL
LIN {X 0,Y 716.599,Z 1009.498,A -85,B 0,C 180,E1 2940.518,E2 2940.518} C_VEL
LIN {X 0,Y 715.1,Z 1050.096,A -85,B 0,C 180,E1 2943.749,E2 2943.749} C_VEL
LIN {X 0,Y 714.108,Z 1082.403,A -85,B 0,C 180,E1 2946.924,E2 2946.924} C_VEL
LIN {X 0,Y 713.277,Z 1111.354,A -85,B 0,C 180,E1 2950.421,E2 2950.421} C_VEL
LIN {X 0,Y 712.841,Z 1134.959,A -85,B 0,C 180,E1 2954.004,E2 2954.004} C_VEL
LIN {X 0,Y 712.485,Z 1153.894,A -85,B 0,C 180,E1 2957.756,E2 2957.756} C_VEL
LIN {X 0,Y 712.372,Z 1167.469,A -85,B 0,C 180,E1 2961.461,E2 2961.461} C_VEL
LIN {X 0,Y 712.284,Z 1175.982,A -85,B 0,C 180,E1 2965.133,E2 2965.133} C_VEL
LIN {X 0,Y 712.226,Z 1179.681,A -85,B 0,C 180,E1 2968.785,E2 2968.785} C_VEL
LIN {X 0,Y 712.254,Z 1178.925,A -85,B 0,C 180,E1 2972.432,E2 2972.432} C_VEL
LIN {X 0,Y 712.336,Z 1173.473,A -85,B 0,C 180,E1 2976.089,E2 2976.089} C_VEL
LIN {X 0,Y 712.373,Z 1163.262,A -85,B 0,C 180,E1 2979.771,E2 2979.771} C_VEL
LIN {X 0,Y 712.542,Z 1147.786,A -85,B 0,C 180,E1 2983.491,E2 2983.491} C_VEL
LIN {X 0,Y 712.883,Z 1128.636,A -85,B 0,C 180,E1 2986.946,E2 2986.946} C_VEL
LIN {X 0,Y 713.514,Z 1102.772,A -85,B 0,C 180,E1 2990.616,E2 2990.616} C_VEL
LIN {X 0,Y 714.398,Z 1071.167,A -85,B 0,C 180,E1 2994.162,E2 2994.162} C_VEL
LIN {X 0,Y 715.591,Z 1036.39,A -85,B 0,C 180,E1 2997.333,E2 2997.333} C_VEL
LIN {X 0,Y 717.22,Z 993.975,A -85,B 0,C 180,E1 3000.445,E2 3000.445} C_VEL
LIN {X 0,Y 718.762,Z 951.302,A -85,B 0,C 180,E1 3002.923,E2 3002.923} C_VEL
LIN {X 0,Y 720.391,Z 906.146,A -85,B 0,C 180,E1 3004.974,E2 3004.974} C_VEL
LIN {X 0,Y 721.59,Z 862.461,A -85,B 0,C 180,E1 3006.463,E2 3006.463} C_VEL
LIN {X 0,Y 722.523,Z 817.457,A -85,B 0,C 180,E1 3007.527,E2 3007.527} C_VEL
LIN {X 0,Y 722.268,Z 782.194,A -85,B 0,C 180,E1 3008.097,E2 3008.097} C_VEL
LIN {X 0,Y 711.984,Z 763.183,A -85,B 0,C 180,E1 3008.992,E2 3008.992} C_VEL
LIN {X 0,Y 711.884,Z 762.06,A -85,B 0,C 180,E1 3009.065,E2 3009.065} C_VEL
LIN {X 0,Y 712.158,Z 762.06,A -85,B 0,C 180,E1 3013.844,E2 3013.844} C_VEL
LIN {X 0,Y 711.901,Z 762.06,A -85,B 0,C 180,E1 3019.832,E2 3019.832} C_VEL
LIN {X 0,Y 711.918,Z 762.06,A -85,B 0,C 180,E1 3025.047,E2 3025.047} C_VEL
LIN {X 0,Y 711.905,Z 762.06,A -85,B 0,C 180,E1 3029.387,E2 3029.387} C_VEL
LIN {X 0,Y 711.917,Z 762.06,A -85,B 0,C 180,E1 3034.891,E2 3034.891} C_VEL
LIN {X 0,Y 711.923,Z 762.06,A -85,B 0,C 180,E1 3040.157,E2 3040.157} C_VEL
LIN {X 0,Y 712.024,Z 762.06,A -85,B 0,C 180,E1 3045.255,E2 3045.255} C_VEL
LIN {X 0,Y 712.251,Z 762.06,A -85,B 0,C 180,E1 3050.236,E2 3050.236} C_VEL
LIN {X 0,Y 712.213,Z 762.06,A -85,B 0,C 180,E1 3055.139,E2 3055.139} C_VEL
LIN {X 0,Y 712.32,Z 762.06,A -85,B 0,C 180,E1 3060.007,E2 3060.007} C_VEL
LIN {X 0,Y 712.385,Z 762.06,A -85,B 0,C 180,E1 3064.874,E2 3064.874} C_VEL
LIN {X 0,Y 712.175,Z 762.06,A -85,B 0,C 180,E1 3069.779,E2 3069.779} C_VEL
LIN {X 0,Y 712.125,Z 762.06,A -85,B 0,C 180,E1 3071.671,E2 3071.671} C_VEL
LIN {X 0,Y 710.892,Z 762.06,A -85,B 0,C 180,E1 3072.366,E2 3072.366} C_VEL
LIN {X 0,Y 704.284,Z 762.06,A -85,B 0,C 180,E1 3074.254,E2 3074.254} C_VEL
LIN {X 0,Y 704.194,Z 762.06,A -85,B 0,C 180,E1 3074.432,E2 3074.432} C_VEL
LIN {X 0,Y 704.267,Z 762.06,A -85,B 0,C 180,E1 3079.249,E2 3079.249} C_VEL
LIN {X 0,Y 704.225,Z 762.06,A -85,B 0,C 180,E1 3084.065,E2 3084.065} C_VEL
LIN {X 0,Y 704.114,Z 762.06,A -85,B 0,C 180,E1 3089.582,E2 3089.582} C_VEL
LIN {X 0,Y 704.079,Z 762.06,A -85,B 0,C 180,E1 3093.923,E2 3093.923} C_VEL
LIN {X 0,Y 703.939,Z 762.06,A -85,B 0,C 180,E1 3098.504,E2 3098.504} C_VEL
LIN {X 0,Y 704.237,Z 762.06,A -85,B 0,C 180,E1 3103.367,E2 3103.367} C_VEL
LIN {X 0,Y 704.004,Z 762.06,A -85,B 0,C 180,E1 3108.702,E2 3108.702} C_VEL
LIN {X 0,Y 704.162,Z 762.737,A -85,B 0,C 180,E1 3110.05,E2 3110.05} C_VEL
LIN {X 0,Y 716.538,Z 786.205,A -85,B 0,C 180,E1 3111.17,E2 3111.17} C_VEL
LIN {X 0,Y 716.19,Z 851.328,A -85,B 0,C 180,E1 3112.115,E2 3112.115} C_VEL
LIN {X 0,Y 714.856,Z 896.002,A -85,B 0,C 180,E1 3113.199,E2 3113.199} C_VEL
LIN {X 0,Y 713.173,Z 945.101,A -85,B 0,C 180,E1 3114.965,E2 3114.965} C_VEL
LIN {X 0,Y 711.453,Z 989.806,A -85,B 0,C 180,E1 3117.113,E2 3117.113} C_VEL
LIN {X 0,Y 709.685,Z 1034.039,A -85,B 0,C 180,E1 3119.861,E2 3119.861} C_VEL
LIN {X 0,Y 708.04,Z 1072.491,A -85,B 0,C 180,E1 3122.833,E2 3122.833} C_VEL
LIN {X 0,Y 706.734,Z 1108.5,A -85,B 0,C 180,E1 3126.279,E2 3126.279} C_VEL
LIN {X 0,Y 705.626,Z 1139.232,A -85,B 0,C 180,E1 3129.961,E2 3129.961} C_VEL
LIN {X 0,Y 705.069,Z 1162.847,A -85,B 0,C 180,E1 3133.502,E2 3133.502} C_VEL
LIN {X 0,Y 704.694,Z 1181.717,A -85,B 0,C 180,E1 3137.156,E2 3137.156} C_VEL
LIN {X 0,Y 704.575,Z 1196.148,A -85,B 0,C 180,E1 3140.971,E2 3140.971} C_VEL
LIN {X 0,Y 704.442,Z 1204.797,A -85,B 0,C 180,E1 3144.46,E2 3144.46} C_VEL
LIN {X 0,Y 704.499,Z 1208.96,A -85,B 0,C 180,E1 3147.541,E2 3147.541} C_VEL
LIN {X 0,Y 704.634,Z 1209.669,A -85,B 0,C 180,E1 3151.228,E2 3151.228} C_VEL
LIN {X 0,Y 704.43,Z 1205.912,A -85,B 0,C 180,E1 3154.922,E2 3154.922} C_VEL
LIN {X 0,Y 704.413,Z 1197.334,A -85,B 0,C 180,E1 3158.636,E2 3158.636} C_VEL
LIN {X 0,Y 704.539,Z 1185.05,A -85,B 0,C 180,E1 3162.07,E2 3162.07} C_VEL
LIN {X 0,Y 704.88,Z 1167.523,A -85,B 0,C 180,E1 3165.671,E2 3165.671} C_VEL
LIN {X 0,Y 705.495,Z 1144.438,A -85,B 0,C 180,E1 3169.336,E2 3169.336} C_VEL
LIN {X 0,Y 706.312,Z 1116.161,A -85,B 0,C 180,E1 3172.875,E2 3172.875} C_VEL
LIN {X 0,Y 707.636,Z 1082.966,A -85,B 0,C 180,E1 3176.247,E2 3176.247} C_VEL
LIN {X 0,Y 709.234,Z 1043.383,A -85,B 0,C 180,E1 3179.477,E2 3179.477} C_VEL
LIN {X 0,Y 710.956,Z 1003.581,A -85,B 0,C 180,E1 3182.097,E2 3182.097} C_VEL
LIN {X 0,Y 712.833,Z 959.309,A -85,B 0,C 180,E1 3184.402,E2 3184.402} C_VEL
LIN {X 0,Y 714.436,Z 915.93,A -85,B 0,C 180,E1 3186.147,E2 3186.147} C_VEL
LIN {X 0,Y 715.674,Z 871.198,A -85,B 0,C 180,E1 3187.456,E2 3187.456} C_VEL
LIN {X 0,Y 716.505,Z 826.331,A -85,B 0,C 180,E1 3188.31,E2 3188.31} C_VEL
LIN {X 0,Y 716.063,Z 785.504,A -85,B 0,C 180,E1 3188.869,E2 3188.869} C_VEL
LIN {X 0,Y 703.99,Z 763.11,A -85,B 0,C 180,E1 3189.957,E2 3189.957} C_VEL
LIN {X 0,Y 703.903,Z 762.06,A -85,B 0,C 180,E1 3190.092,E2 3190.092} C_VEL
LIN {X 0,Y 704.205,Z 762.06,A -85,B 0,C 180,E1 3195.082,E2 3195.082} C_VEL
LIN {X 0,Y 704.047,Z 762.06,A -85,B 0,C 180,E1 3200.594,E2 3200.594} C_VEL
LIN {X 0,Y 703.974,Z 762.06,A -85,B 0,C 180,E1 3206.072,E2 3206.072} C_VEL
LIN {X 0,Y 704.001,Z 762.06,A -85,B 0,C 180,E1 3210.413,E2 3210.413} C_VEL
LIN {X 0,Y 704.067,Z 762.06,A -85,B 0,C 180,E1 3214.575,E2 3214.575} C_VEL
LIN {X 0,Y 704.041,Z 762.06,A -85,B 0,C 180,E1 3219.91,E2 3219.91} C_VEL
LIN {X 0,Y 704.23,Z 762.06,A -85,B 0,C 180,E1 3225.073,E2 3225.073} C_VEL
LIN {X 0,Y 704.281,Z 762.06,A -85,B 0,C 180,E1 3230.11,E2 3230.11} C_VEL
LIN {X 0,Y 704.505,Z 762.06,A -85,B 0,C 180,E1 3235.072,E2 3235.072} C_VEL
LIN {X 0,Y 704.39,Z 762.06,A -85,B 0,C 180,E1 3239.993,E2 3239.993} C_VEL
LIN {X 0,Y 704.361,Z 762.06,A -85,B 0,C 180,E1 3244.915,E2 3244.915} C_VEL
LIN {X 0,Y 704.336,Z 762.06,A -85,B 0,C 180,E1 3249.874,E2 3249.874} C_VEL
LIN {X 0,Y 704.031,Z 762.06,A -85,B 0,C 180,E1 3255.015,E2 3255.015} C_VEL
LIN {X 0,Y 704.035,Z 762.06,A -85,B 0,C 180,E1 3260.075,E2 3260.075} C_VEL
LIN {X 0,Y 704.03,Z 762.06,A -85,B 0,C 180,E1 3265.41,E2 3265.41} C_VEL
LIN {X 0,Y 704.003,Z 762.06,A -85,B 0,C 180,E1 3270.844,E2 3270.844} C_VEL
LIN {X 0,Y 704.041,Z 762.06,A -85,B 0,C 180,E1 3275.402,E2 3275.402} C_VEL
LIN {X 0,Y 703.854,Z 762.06,A -85,B 0,C 180,E1 3280.081,E2 3280.081} C_VEL
LIN {X 0,Y 703.86,Z 762.06,A -85,B 0,C 180,E1 3285.094,E2 3285.094} C_VEL
LIN {X 0,Y 704.29,Z 762.06,A -85,B 0,C 180,E1 3290.219,E2 3290.219} C_VEL
LIN {X 0,Y 704.29,Z 762.06,A -85,B 0,C 180,E1 3290.384,E2 3290.384} C_VEL
LIN {X 0,Y 708.664,Z 771.834,A -85,B 0,C 180,E1 3290.811,E2 3290.811} C_VEL
LIN {X 0,Y 716.659,Z 786.687,A -85,B 0,C 180,E1 3291.517,E2 3291.517} C_VEL
LIN {X 0,Y 715.935,Z 832.859,A -85,B 0,C 180,E1 3292.311,E2 3292.311} C_VEL
LIN {X 0,Y 714.51,Z 879.641,A -85,B 0,C 180,E1 3293.596,E2 3293.596} C_VEL
LIN {X 0,Y 712.978,Z 924.856,A -85,B 0,C 180,E1 3295.345,E2 3295.345} C_VEL
LIN {X 0,Y 711.063,Z 970.785,A -85,B 0,C 180,E1 3297.698,E2 3297.698} C_VEL
LIN {X 0,Y 709.294,Z 1012.106,A -85,B 0,C 180,E1 3300.384,E2 3300.384} C_VEL
LIN {X 0,Y 707.629,Z 1051.923,A -85,B 0,C 180,E1 3303.614,E2 3303.614} C_VEL
LIN {X 0,Y 706.325,Z 1086.364,A -85,B 0,C 180,E1 3307.103,E2 3307.103} C_VEL
LIN {X 0,Y 705.443,Z 1114.879,A -85,B 0,C 180,E1 3310.682,E2 3310.682} C_VEL
LIN {X 0,Y 704.929,Z 1137.644,A -85,B 0,C 180,E1 3314.307,E2 3314.307} C_VEL
LIN {X 0,Y 704.599,Z 1155.244,A -85,B 0,C 180,E1 3317.931,E2 3317.931} C_VEL
LIN {X 0,Y 704.492,Z 1167.468,A -85,B 0,C 180,E1 3321.365,E2 3321.365} C_VEL
LIN {X 0,Y 704.39,Z 1175.981,A -85,B 0,C 180,E1 3325.078,E2 3325.078} C_VEL
LIN {X 0,Y 704.326,Z 1179.681,A -85,B 0,C 180,E1 3328.771,E2 3328.771} C_VEL
LIN {X 0,Y 704.37,Z 1178.922,A -85,B 0,C 180,E1 3332.46,E2 3332.46} C_VEL
LIN {X 0,Y 704.434,Z 1173.474,A -85,B 0,C 180,E1 3336.158,E2 3336.158} C_VEL
LIN {X 0,Y 704.508,Z 1163.264,A -85,B 0,C 180,E1 3339.881,E2 3339.881} C_VEL
LIN {X 0,Y 704.704,Z 1147.79,A -85,B 0,C 180,E1 3343.644,E2 3343.644} C_VEL
LIN {X 0,Y 705.078,Z 1128.641,A -85,B 0,C 180,E1 3347.139,E2 3347.139} C_VEL
LIN {X 0,Y 705.771,Z 1104.026,A -85,B 0,C 180,E1 3350.689,E2 3350.689} C_VEL
LIN {X 0,Y 706.798,Z 1073.729,A -85,B 0,C 180,E1 3354.172,E2 3354.172} C_VEL
LIN {X 0,Y 708.165,Z 1038.723,A -85,B 0,C 180,E1 3357.452,E2 3357.452} C_VEL
LIN {X 0,Y 709.946,Z 997.034,A -85,B 0,C 180,E1 3360.576,E2 3360.576} C_VEL
LIN {X 0,Y 711.797,Z 955.297,A -85,B 0,C 180,E1 3363.072,E2 3363.072} C_VEL
LIN {X 0,Y 713.531,Z 911.291,A -85,B 0,C 180,E1 3365.137,E2 3365.137} C_VEL
LIN {X 0,Y 714.968,Z 867.774,A -85,B 0,C 180,E1 3366.689,E2 3366.689} C_VEL
LIN {X 0,Y 716.112,Z 822.418,A -85,B 0,C 180,E1 3367.822,E2 3367.822} C_VEL
LIN {X 0,Y 716.071,Z 785.386,A -85,B 0,C 180,E1 3368.448,E2 3368.448} C_VEL
LIN {X 0,Y 704.05,Z 763.29,A -85,B 0,C 180,E1 3369.516,E2 3369.516} C_VEL
LIN {X 0,Y 703.967,Z 762.06,A -85,B 0,C 180,E1 3369.598,E2 3369.598} C_VEL
LIN {X 0,Y 704.236,Z 762.06,A -85,B 0,C 180,E1 3373.365,E2 3373.365} C_VEL
LIN {X 0,Y 703.938,Z 762.06,A -85,B 0,C 180,E1 3378.707,E2 3378.707} C_VEL
LIN {X 0,Y 703.964,Z 762.06,A -85,B 0,C 180,E1 3383.07,E2 3383.07} C_VEL
LIN {X 0,Y 703.938,Z 762.06,A -85,B 0,C 180,E1 3387.556,E2 3387.556} C_VEL
LIN {X 0,Y 703.896,Z 762.06,A -85,B 0,C 180,E1 3391.829,E2 3391.829} C_VEL
LIN {X 0,Y 703.894,Z 762.06,A -85,B 0,C 180,E1 3395.939,E2 3395.939} C_VEL
LIN {X 0,Y 703.922,Z 762.06,A -85,B 0,C 180,E1 3400.832,E2 3400.832} C_VEL
LIN {X 0,Y 704.136,Z 762.06,A -85,B 0,C 180,E1 3406.355,E2 3406.355} C_VEL
LIN {X 0,Y 704.252,Z 762.06,A -85,B 0,C 180,E1 3411.37,E2 3411.37} C_VEL
LIN {X 0,Y 704.433,Z 762.06,A -85,B 0,C 180,E1 3416.318,E2 3416.318} C_VEL
LIN {X 0,Y 704.573,Z 762.06,A -85,B 0,C 180,E1 3421.236,E2 3421.236} C_VEL
LIN {X 0,Y 704.277,Z 762.06,A -85,B 0,C 180,E1 3426.165,E2 3426.165} C_VEL
LIN {X 0,Y 704.227,Z 762.06,A -85,B 0,C 180,E1 3431.141,E2 3431.141} C_VEL
LIN {X 0,Y 704.194,Z 762.06,A -85,B 0,C 180,E1 3434.432,E2 3434.432} C_VEL
LIN {X 0,Y 700.282,Z 762.06,A -85,B 0,C 180,E1 3435.822,E2 3435.822} C_VEL
LIN {X 0,Y 696.42,Z 762.06,A -85,B 0,C 180,E1 3437.229,E2 3437.229} C_VEL
LIN {X 0,Y 696.286,Z 762.06,A -85,B 0,C 180,E1 3441.655,E2 3441.655} C_VEL
LIN {X 0,Y 696.24,Z 762.06,A -85,B 0,C 180,E1 3445.731,E2 3445.731} C_VEL
LIN {X 0,Y 696.179,Z 762.06,A -85,B 0,C 180,E1 3449.953,E2 3449.953} C_VEL
LIN {X 0,Y 696.11,Z 762.06,A -85,B 0,C 180,E1 3454.42,E2 3454.42} C_VEL
LIN {X 0,Y 696.006,Z 762.06,A -85,B 0,C 180,E1 3459.026,E2 3459.026} C_VEL
LIN {X 0,Y 696.252,Z 762.06,A -85,B 0,C 180,E1 3464.256,E2 3464.256} C_VEL
LIN {X 0,Y 696.137,Z 762.06,A -85,B 0,C 180,E1 3469.484,E2 3469.484} C_VEL
LIN {X 0,Y 700.314,Z 771.304,A -85,B 0,C 180,E1 3469.898,E2 3469.898} C_VEL
LIN {X 0,Y 710.45,Z 789.392,A -85,B 0,C 180,E1 3470.815,E2 3470.815} C_VEL
LIN {X 0,Y 709.913,Z 852.545,A -85,B 0,C 180,E1 3471.746,E2 3471.746} C_VEL
LIN {X 0,Y 708.37,Z 897.912,A -85,B 0,C 180,E1 3472.871,E2 3472.871} C_VEL
LIN {X 0,Y 706.456,Z 947.125,A -85,B 0,C 180,E1 3474.672,E2 3474.672} C_VEL
LIN {X 0,Y 704.462,Z 991.661,A -85,B 0,C 180,E1 3476.855,E2 3476.855} C_VEL
LIN {X 0,Y 702.451,Z 1036.155,A -85,B 0,C 180,E1 3479.668,E2 3479.668} C_VEL
LIN {X 0,Y 700.564,Z 1074.564,A -85,B 0,C 180,E1 3482.707,E2 3482.707} C_VEL
LIN {X 0,Y 699.137,Z 1109.279,A -85,B 0,C 180,E1 3486.089,E2 3486.089} C_VEL
LIN {X 0,Y 697.89,Z 1140.365,A -85,B 0,C 180,E1 3489.883,E2 3489.883} C_VEL
LIN {X 0,Y 697.218,Z 1164.706,A -85,B 0,C 180,E1 3493.634,E2 3493.634} C_VEL
LIN {X 0,Y 696.765,Z 1183.695,A -85,B 0,C 180,E1 3497.474,E2 3497.474} C_VEL
LIN {X 0,Y 696.711,Z 1196.145,A -85,B 0,C 180,E1 3500.868,E2 3500.868} C_VEL
LIN {X 0,Y 696.561,Z 1204.797,A -85,B 0,C 180,E1 3504.397,E2 3504.397} C_VEL
LIN {X 0,Y 696.596,Z 1208.957,A -85,B 0,C 180,E1 3507.513,E2 3507.513} C_VEL
LIN {X 0,Y 696.732,Z 1209.669,A -85,B 0,C 180,E1 3511.242,E2 3511.242} C_VEL
LIN {X 0,Y 696.541,Z 1205.912,A -85,B 0,C 180,E1 3514.978,E2 3514.978} C_VEL
LIN {X 0,Y 696.564,Z 1197.334,A -85,B 0,C 180,E1 3518.734,E2 3518.734} C_VEL
LIN {X 0,Y 696.689,Z 1185.051,A -85,B 0,C 180,E1 3522.208,E2 3522.208} C_VEL
LIN {X 0,Y 697.042,Z 1167.245,A -85,B 0,C 180,E1 3525.903,E2 3525.903} C_VEL
LIN {X 0,Y 697.739,Z 1144.942,A -85,B 0,C 180,E1 3529.485,E2 3529.485} C_VEL
LIN {X 0,Y 698.723,Z 1116.163,A -85,B 0,C 180,E1 3533.138,E2 3533.138} C_VEL
LIN {X 0,Y 700.257,Z 1081.866,A -85,B 0,C 180,E1 3536.646,E2 3536.646} C_VEL
LIN {X 0,Y 702.133,Z 1041.905,A -85,B 0,C 180,E1 3539.919,E2 3539.919} C_VEL
LIN {X 0,Y 704.078,Z 1001.052,A -85,B 0,C 180,E1 3542.601,E2 3542.601} C_VEL
LIN {X 0,Y 706.261,Z 956.125,A -85,B 0,C 180,E1 3544.924,E2 3544.924} C_VEL
LIN {X 0,Y 708.01,Z 913.615,A -85,B 0,C 180,E1 3546.611,E2 3546.611} C_VEL
LIN {X 0,Y 709.389,Z 870.223,A -85,B 0,C 180,E1 3547.871,E2 3547.871} C_VEL
LIN {X 0,Y 710.325,Z 824.022,A -85,B 0,C 180,E1 3548.74,E2 3548.74} C_VEL
LIN {X 0,Y 709.835,Z 788.415,A -85,B 0,C 180,E1 3549.238,E2 3549.238} C_VEL
LIN {X 0,Y 696.057,Z 762.871,A -85,B 0,C 180,E1 3550.51,E2 3550.51} C_VEL
LIN {X 0,Y 696.195,Z 762.06,A -85,B 0,C 180,E1 3552.438,E2 3552.438} C_VEL
LIN {X 0,Y 696.039,Z 762.06,A -85,B 0,C 180,E1 3557.697,E2 3557.697} C_VEL
LIN {X 0,Y 696.06,Z 762.06,A -85,B 0,C 180,E1 3562.561,E2 3562.561} C_VEL
LIN {X 0,Y 696.018,Z 762.06,A -85,B 0,C 180,E1 3567.856,E2 3567.856} C_VEL
LIN {X 0,Y 696.111,Z 762.06,A -85,B 0,C 180,E1 3572.875,E2 3572.875} C_VEL
LIN {X 0,Y 696.075,Z 762.06,A -85,B 0,C 180,E1 3576.993,E2 3576.993} C_VEL
LIN {X 0,Y 696.316,Z 762.06,A -85,B 0,C 180,E1 3582.718,E2 3582.718} C_VEL
LIN {X 0,Y 696.383,Z 762.06,A -85,B 0,C 180,E1 3587.544,E2 3587.544} C_VEL
LIN {X 0,Y 696.367,Z 762.06,A -85,B 0,C 180,E1 3592.513,E2 3592.513} C_VEL
LIN {X 0,Y 696.457,Z 762.06,A -85,B 0,C 180,E1 3596.426,E2 3596.426} C_VEL
LIN {X 0,Y 696.49,Z 762.06,A -85,B 0,C 180,E1 3599.993,E2 3599.993} C_VEL
LIN {X 0,Y 696.48,Z 762.06,A -85,B 0,C 180,E1 3604.971,E2 3604.971} C_VEL
LIN {X 0,Y 696.419,Z 762.06,A -85,B 0,C 180,E1 3609.988,E2 3609.988} C_VEL
LIN {X 0,Y 696.129,Z 762.06,A -85,B 0,C 180,E1 3615.09,E2 3615.09} C_VEL
LIN {X 0,Y 696.146,Z 762.06,A -85,B 0,C 180,E1 3621.032,E2 3621.032} C_VEL
LIN {X 0,Y 696.103,Z 762.06,A -85,B 0,C 180,E1 3625.721,E2 3625.721} C_VEL
LIN {X 0,Y 696.078,Z 762.06,A -85,B 0,C 180,E1 3629.942,E2 3629.942} C_VEL
LIN {X 0,Y 696.096,Z 762.06,A -85,B 0,C 180,E1 3634.421,E2 3634.421} C_VEL
LIN {X 0,Y 695.997,Z 762.06,A -85,B 0,C 180,E1 3639.008,E2 3639.008} C_VEL
LIN {X 0,Y 695.916,Z 762.06,A -85,B 0,C 180,E1 3644.23,E2 3644.23} C_VEL
LIN {X 0,Y 696.357,Z 762.06,A -85,B 0,C 180,E1 3649.794,E2 3649.794} C_VEL
LIN {X 0,Y 704.026,Z 777.524,A -85,B 0,C 180,E1 3650.577,E2 3650.577} C_VEL
LIN {X 0,Y 710.439,Z 789.724,A -85,B 0,C 180,E1 3651.16,E2 3651.16} C_VEL
LIN {X 0,Y 709.566,Z 835.325,A -85,B 0,C 180,E1 3651.975,E2 3651.975} C_VEL
LIN {X 0,Y 707.999,Z 881.01,A -85,B 0,C 180,E1 3653.254,E2 3653.254} C_VEL
LIN {X 0,Y 706.185,Z 926.905,A -85,B 0,C 180,E1 3655.065,E2 3655.065} C_VEL
LIN {X 0,Y 704.034,Z 972.59,A -85,B 0,C 180,E1 3657.444,E2 3657.444} C_VEL
LIN {X 0,Y 702.071,Z 1012.382,A -85,B 0,C 180,E1 3660.07,E2 3660.07} C_VEL
LIN {X 0,Y 700.23,Z 1052.222,A -85,B 0,C 180,E1 3663.341,E2 3663.341} C_VEL
LIN {X 0,Y 698.699,Z 1086.36,A -85,B 0,C 180,E1 3666.839,E2 3666.839} C_VEL
LIN {X 0,Y 697.699,Z 1115.055,A -85,B 0,C 180,E1 3670.486,E2 3670.486} C_VEL
LIN {X 0,Y 697.077,Z 1138.577,A -85,B 0,C 180,E1 3674.297,E2 3674.297} C_VEL
LIN {X 0,Y 696.753,Z 1155.243,A -85,B 0,C 180,E1 3677.793,E2 3677.793} C_VEL
LIN {X 0,Y 696.629,Z 1167.466,A -85,B 0,C 180,E1 3681.267,E2 3681.267} C_VEL
LIN {X 0,Y 696.495,Z 1175.98,A -85,B 0,C 180,E1 3685.022,E2 3685.022} C_VEL
LIN {X 0,Y 696.425,Z 1179.681,A -85,B 0,C 180,E1 3688.757,E2 3688.757} C_VEL
LIN {X 0,Y 696.469,Z 1178.92,A -85,B 0,C 180,E1 3692.488,E2 3692.488} C_VEL
LIN {X 0,Y 696.548,Z 1173.475,A -85,B 0,C 180,E1 3696.228,E2 3696.228} C_VEL
LIN {X 0,Y 696.613,Z 1163.265,A -85,B 0,C 180,E1 3699.994,E2 3699.994} C_VEL
LIN {X 0,Y 696.874,Z 1147.794,A -85,B 0,C 180,E1 3703.8,E2 3703.8} C_VEL
LIN {X 0,Y 697.34,Z 1127.074,A -85,B 0,C 180,E1 3707.595,E2 3707.595} C_VEL
LIN {X 0,Y 698.099,Z 1101.927,A -85,B 0,C 180,E1 3711.199,E2 3711.199} C_VEL
LIN {X 0,Y 699.451,Z 1069.531,A -85,B 0,C 180,E1 3714.887,E2 3714.887} C_VEL
LIN {X 0,Y 700.984,Z 1035.414,A -85,B 0,C 180,E1 3718.035,E2 3718.035} C_VEL
LIN {X 0,Y 703.028,Z 993.388,A -85,B 0,C 180,E1 3721.17,E2 3721.17} C_VEL
LIN {X 0,Y 705.135,Z 949.156,A -85,B 0,C 180,E1 3723.762,E2 3723.762} C_VEL
LIN {X 0,Y 707.227,Z 904.49,A -85,B 0,C 180,E1 3725.798,E2 3725.798} C_VEL
LIN {X 0,Y 708.826,Z 861.116,A -85,B 0,C 180,E1 3727.272,E2 3727.272} C_VEL
LIN {X 0,Y 709.996,Z 817.775,A -85,B 0,C 180,E1 3728.301,E2 3728.301} C_VEL
LIN {X 0,Y 709.853,Z 788.344,A -85,B 0,C 180,E1 3728.807,E2 3728.807} C_VEL
LIN {X 0,Y 696.173,Z 763.48,A -85,B 0,C 180,E1 3730.051,E2 3730.051} C_VEL
LIN {X 0,Y 696.054,Z 762.06,A -85,B 0,C 180,E1 3730.132,E2 3730.132} C_VEL
LIN {X 0,Y 696.23,Z 762.06,A -85,B 0,C 180,E1 3734.273,E2 3734.273} C_VEL
LIN {X 0,Y 696.065,Z 762.06,A -85,B 0,C 180,E1 3739.45,E2 3739.45} C_VEL
LIN {X 0,Y 696.029,Z 762.06,A -85,B 0,C 180,E1 3744.128,E2 3744.128} C_VEL
LIN {X 0,Y 696.032,Z 762.06,A -85,B 0,C 180,E1 3748.61,E2 3748.61} C_VEL
LIN {X 0,Y 696.092,Z 762.06,A -85,B 0,C 180,E1 3754.279,E2 3754.279} C_VEL
LIN {X 0,Y 696.071,Z 762.06,A -85,B 0,C 180,E1 3759.685,E2 3759.685} C_VEL
LIN {X 0,Y 696.15,Z 762.06,A -85,B 0,C 180,E1 3764.911,E2 3764.911} C_VEL
LIN {X 0,Y 696.433,Z 762.06,A -85,B 0,C 180,E1 3770.012,E2 3770.012} C_VEL
LIN {X 0,Y 696.421,Z 762.06,A -85,B 0,C 180,E1 3775.029,E2 3775.029} C_VEL
LIN {X 0,Y 696.52,Z 762.06,A -85,B 0,C 180,E1 3780.007,E2 3780.007} C_VEL
LIN {X 0,Y 696.562,Z 762.06,A -85,B 0,C 180,E1 3784.985,E2 3784.985} C_VEL
LIN {X 0,Y 696.37,Z 762.06,A -85,B 0,C 180,E1 3790.003,E2 3790.003} C_VEL
LIN {X 0,Y 696.348,Z 762.06,A -85,B 0,C 180,E1 3795.1,E2 3795.1} C_VEL
LIN {X 0,Y 696.42,Z 762.06,A -85,B 0,C 180,E1 3797.229,E2 3797.229} C_VEL
LIN {X 0,Y 693.909,Z 762.06,A -85,B 0,C 180,E1 3798.287,E2 3798.287} C_VEL
LIN {X 0,Y 688.48,Z 762.06,A -85,B 0,C 180,E1 3799.867,E2 3799.867} C_VEL
LIN {X 0,Y 688.385,Z 762.06,A -85,B 0,C 180,E1 3800.05,E2 3800.05} C_VEL
LIN {X 0,Y 688.337,Z 762.06,A -85,B 0,C 180,E1 3804.657,E2 3804.657} C_VEL
LIN {X 0,Y 688.301,Z 762.06,A -85,B 0,C 180,E1 3808.885,E2 3808.885} C_VEL
LIN {X 0,Y 688.221,Z 762.06,A -85,B 0,C 180,E1 3813.45,E2 3813.45} C_VEL
LIN {X 0,Y 688.145,Z 762.06,A -85,B 0,C 180,E1 3817.945,E2 3817.945} C_VEL
LIN {X 0,Y 688.309,Z 762.06,A -85,B 0,C 180,E1 3823.573,E2 3823.573} C_VEL
LIN {X 0,Y 688.178,Z 762.255,A -85,B 0,C 180,E1 3828.919,E2 3828.919} C_VEL
LIN {X 0,Y 692.539,Z 771.551,A -85,B 0,C 180,E1 3829.358,E2 3829.358} C_VEL
LIN {X 0,Y 704.317,Z 792.711,A -85,B 0,C 180,E1 3830.45,E2 3830.45} C_VEL
LIN {X 0,Y 703.663,Z 853.846,A -85,B 0,C 180,E1 3831.371,E2 3831.371} C_VEL
LIN {X 0,Y 701.94,Z 898.747,A -85,B 0,C 180,E1 3832.502,E2 3832.502} C_VEL
LIN {X 0,Y 699.814,Z 948.261,A -85,B 0,C 180,E1 3834.337,E2 3834.337} C_VEL
LIN {X 0,Y 697.517,Z 993.448,A -85,B 0,C 180,E1 3836.591,E2 3836.591} C_VEL
LIN {X 0,Y 695.227,Z 1038.233,A -85,B 0,C 180,E1 3839.47,E2 3839.47} C_VEL
LIN {X 0,Y 693.043,Z 1077.404,A -85,B 0,C 180,E1 3842.646,E2 3842.646} C_VEL
LIN {X 0,Y 691.518,Z 1110.712,A -85,B 0,C 180,E1 3845.974,E2 3845.974} C_VEL
LIN {X 0,Y 690.179,Z 1140.983,A -85,B 0,C 180,E1 3849.733,E2 3849.733} C_VEL
LIN {X 0,Y 689.43,Z 1164.708,A -85,B 0,C 180,E1 3853.444,E2 3853.444} C_VEL
LIN {X 0,Y 688.908,Z 1183.696,A -85,B 0,C 180,E1 3857.329,E2 3857.329} C_VEL
LIN {X 0,Y 688.728,Z 1197.33,A -85,B 0,C 180,E1 3861.165,E2 3861.165} C_VEL
LIN {X 0,Y 688.643,Z 1205.91,A -85,B 0,C 180,E1 3864.964,E2 3864.964} C_VEL
LIN {X 0,Y 688.571,Z 1209.668,A -85,B 0,C 180,E1 3868.742,E2 3868.742} C_VEL
LIN {X 0,Y 688.769,Z 1208.956,A -85,B 0,C 180,E1 3872.514,E2 3872.514} C_VEL
LIN {X 0,Y 688.74,Z 1203.571,A -85,B 0,C 180,E1 3876.297,E2 3876.297} C_VEL
LIN {X 0,Y 688.901,Z 1192.319,A -85,B 0,C 180,E1 3880.425,E2 3880.425} C_VEL
LIN {X 0,Y 689.18,Z 1174.917,A -85,B 0,C 180,E1 3884.604,E2 3884.604} C_VEL
LIN {X 0,Y 689.775,Z 1152.86,A -85,B 0,C 180,E1 3888.521,E2 3888.521} C_VEL
LIN {X 0,Y 690.835,Z 1125.141,A -85,B 0,C 180,E1 3892.336,E2 3892.336} C_VEL
LIN {X 0,Y 692.24,Z 1094.878,A -85,B 0,C 180,E1 3895.696,E2 3895.696} C_VEL
LIN {X 0,Y 694.249,Z 1055.77,A -85,B 0,C 180,E1 3899.196,E2 3899.196} C_VEL
LIN {X 0,Y 696.39,Z 1016.064,A -85,B 0,C 180,E1 3902.037,E2 3902.037} C_VEL
LIN {X 0,Y 698.702,Z 973.393,A -85,B 0,C 180,E1 3904.479,E2 3904.479} C_VEL
LIN {X 0,Y 700.829,Z 928.955,A -85,B 0,C 180,E1 3906.444,E2 3906.444} C_VEL
LIN {X 0,Y 702.702,Z 880.48,A -85,B 0,C 180,E1 3908.016,E2 3908.016} C_VEL
LIN {X 0,Y 704.005,Z 833.344,A -85,B 0,C 180,E1 3909.007,E2 3909.007} C_VEL
LIN {X 0,Y 704.001,Z 792.103,A -85,B 0,C 180,E1 3909.58,E2 3909.58} C_VEL
LIN {X 0,Y 688.29,Z 763.623,A -85,B 0,C 180,E1 3911.054,E2 3911.054} C_VEL
LIN {X 0,Y 688.112,Z 762.06,A -85,B 0,C 180,E1 3911.208,E2 3911.208} C_VEL
LIN {X 0,Y 688.266,Z 762.06,A -85,B 0,C 180,E1 3915.363,E2 3915.363} C_VEL
LIN {X 0,Y 688.159,Z 762.06,A -85,B 0,C 180,E1 3920.443,E2 3920.443} C_VEL
LIN {X 0,Y 688.123,Z 762.06,A -85,B 0,C 180,E1 3925.179,E2 3925.179} C_VEL
LIN {X 0,Y 688.132,Z 762.06,A -85,B 0,C 180,E1 3929.66,E2 3929.66} C_VEL
LIN {X 0,Y 688.252,Z 762.06,A -85,B 0,C 180,E1 3934.181,E2 3934.181} C_VEL
LIN {X 0,Y 688.224,Z 762.06,A -85,B 0,C 180,E1 3939.428,E2 3939.428} C_VEL
LIN {X 0,Y 688.446,Z 762.06,A -85,B 0,C 180,E1 3944.966,E2 3944.966} C_VEL
LIN {X 0,Y 688.463,Z 762.06,A -85,B 0,C 180,E1 3949.881,E2 3949.881} C_VEL
LIN {X 0,Y 688.668,Z 762.06,A -85,B 0,C 180,E1 3954.958,E2 3954.958} C_VEL
LIN {X 0,Y 688.614,Z 762.06,A -85,B 0,C 180,E1 3959.993,E2 3959.993} C_VEL
LIN {X 0,Y 688.575,Z 762.06,A -85,B 0,C 180,E1 3965.028,E2 3965.028} C_VEL
LIN {X 0,Y 688.509,Z 762.06,A -85,B 0,C 180,E1 3970.104,E2 3970.104} C_VEL
LIN {X 0,Y 688.195,Z 762.06,A -85,B 0,C 180,E1 3975.268,E2 3975.268} C_VEL
LIN {X 0,Y 688.228,Z 762.06,A -85,B 0,C 180,E1 3980.557,E2 3980.557} C_VEL
LIN {X 0,Y 688.206,Z 762.06,A -85,B 0,C 180,E1 3985.811,E2 3985.811} C_VEL
LIN {X 0,Y 688.145,Z 762.06,A -85,B 0,C 180,E1 3991.086,E2 3991.086} C_VEL
LIN {X 0,Y 688.161,Z 762.06,A -85,B 0,C 180,E1 3996.348,E2 3996.348} C_VEL
LIN {X 0,Y 688,Z 762.06,A -85,B 0,C 180,E1 4001.69,E2 4001.69} C_VEL
LIN {X 0,Y 688.19,Z 762.06,A -85,B 0,C 180,E1 4007.103,E2 4007.103} C_VEL
LIN {X 0,Y 688.439,Z 762.06,A -85,B 0,C 180,E1 4009.274,E2 4009.274} C_VEL
LIN {X 0,Y 693.191,Z 772.268,A -85,B 0,C 180,E1 4009.768,E2 4009.768} C_VEL
LIN {X 0,Y 704.236,Z 793.674,A -85,B 0,C 180,E1 4010.812,E2 4010.812} C_VEL
LIN {X 0,Y 703.199,Z 838.586,A -85,B 0,C 180,E1 4011.65,E2 4011.65} C_VEL
LIN {X 0,Y 701.423,Z 884.936,A -85,B 0,C 180,E1 4012.99,E2 4012.99} C_VEL
LIN {X 0,Y 699.333,Z 930.71,A -85,B 0,C 180,E1 4014.863,E2 4014.863} C_VEL
LIN {X 0,Y 696.988,Z 975.954,A -85,B 0,C 180,E1 4017.279,E2 4017.279} C_VEL
LIN {X 0,Y 694.569,Z 1018.934,A -85,B 0,C 180,E1 4020.229,E2 4020.229} C_VEL
LIN {X 0,Y 692.562,Z 1056.332,A -85,B 0,C 180,E1 4023.424,E2 4023.424} C_VEL
LIN {X 0,Y 691.014,Z 1090,A -85,B 0,C 180,E1 4026.991,E2 4026.991} C_VEL
LIN {X 0,Y 689.887,Z 1117.071,A -85,B 0,C 180,E1 4030.561,E2 4030.561} C_VEL
LIN {X 0,Y 689.218,Z 1140.405,A -85,B 0,C 180,E1 4034.454,E2 4034.454} C_VEL
LIN {X 0,Y 688.806,Z 1157.849,A -85,B 0,C 180,E1 4038.292,E2 4038.292} C_VEL
LIN {X 0,Y 688.693,Z 1169.221,A -85,B 0,C 180,E1 4041.801,E2 4041.801} C_VEL
LIN {X 0,Y 688.603,Z 1175.979,A -85,B 0,C 180,E1 4044.965,E2 4044.965} C_VEL
LIN {X 0,Y 688.552,Z 1179.681,A -85,B 0,C 180,E1 4048.743,E2 4048.743} C_VEL
LIN {X 0,Y 688.568,Z 1178.918,A -85,B 0,C 180,E1 4052.516,E2 4052.516} C_VEL
LIN {X 0,Y 688.65,Z 1173.476,A -85,B 0,C 180,E1 4056.3,E2 4056.3} C_VEL
LIN {X 0,Y 688.744,Z 1163.267,A -85,B 0,C 180,E1 4060.11,E2 4060.11} C_VEL
LIN {X 0,Y 689.047,Z 1147.798,A -85,B 0,C 180,E1 4063.96,E2 4063.96} C_VEL
LIN {X 0,Y 689.508,Z 1127.715,A -85,B 0,C 180,E1 4067.695,E2 4067.695} C_VEL
LIN {X 0,Y 690.381,Z 1103.337,A -85,B 0,C 180,E1 4071.268,E2 4071.268} C_VEL
LIN {X 0,Y 691.797,Z 1071.947,A -85,B 0,C 180,E1 4074.923,E2 4074.923} C_VEL
LIN {X 0,Y 693.631,Z 1036.985,A -85,B 0,C 180,E1 4078.226,E2 4078.226} C_VEL
LIN {X 0,Y 695.883,Z 994.992,A -85,B 0,C 180,E1 4081.411,E2 4081.411} C_VEL
LIN {X 0,Y 698.234,Z 952.702,A -85,B 0,C 180,E1 4083.945,E2 4083.945} C_VEL
LIN {X 0,Y 700.571,Z 907.034,A -85,B 0,C 180,E1 4086.078,E2 4086.078} C_VEL
LIN {X 0,Y 702.282,Z 865.745,A -85,B 0,C 180,E1 4087.535,E2 4087.535} C_VEL
LIN {X 0,Y 703.704,Z 820.477,A -85,B 0,C 180,E1 4088.653,E2 4088.653} C_VEL
LIN {X 0,Y 703.679,Z 791.67,A -85,B 0,C 180,E1 4089.166,E2 4089.166} C_VEL
LIN {X 0,Y 688.234,Z 763.13,A -85,B 0,C 180,E1 4090.614,E2 4090.614} C_VEL
LIN {X 0,Y 688.154,Z 762.06,A -85,B 0,C 180,E1 4090.735,E2 4090.735} C_VEL
LIN {X 0,Y 688.209,Z 762.06,A -85,B 0,C 180,E1 4095.379,E2 4095.379} C_VEL
LIN {X 0,Y 688.13,Z 762.06,A -85,B 0,C 180,E1 4100.46,E2 4100.46} C_VEL
LIN {X 0,Y 688.109,Z 762.06,A -85,B 0,C 180,E1 4105.196,E2 4105.196} C_VEL
LIN {X 0,Y 688.082,Z 762.06,A -85,B 0,C 180,E1 4109.674,E2 4109.674} C_VEL
LIN {X 0,Y 688.203,Z 762.06,A -85,B 0,C 180,E1 4114.192,E2 4114.192} C_VEL
LIN {X 0,Y 688.173,Z 762.06,A -85,B 0,C 180,E1 4119.442,E2 4119.442} C_VEL
LIN {X 0,Y 688.246,Z 762.06,A -85,B 0,C 180,E1 4125.033,E2 4125.033} C_VEL
LIN {X 0,Y 688.524,Z 762.06,A -85,B 0,C 180,E1 4129.896,E2 4129.896} C_VEL
LIN {X 0,Y 688.52,Z 762.06,A -85,B 0,C 180,E1 4134.972,E2 4134.972} C_VEL
